# B&R Automation Studio project TD52 (part 65)

```c
  /* BusCreator: '<Root>/Bus Creator' incorporates:
   *  BusCreator: '<S1>/Bus Creator2'
   *  DataTypeConversion: '<S1>/Data Type Conversion19'
   *  DataTypeConversion: '<S1>/Data Type Conversion7'
   *  Outport: '<Root>/dbg'
   */
  Gen2_ref_Y->dbg.BDC.FF.wg_cd = (real32_T)r;
  Gen2_ref_Y->dbg.BDC.FF.u_tv_ff = (real32_T)rtb_Product4_d;

  /* MinMax: '<S490>/MinMax' incorporates:
   *  DataTypeConversion: '<S43>/Data Type Conversion25'
   */
  if ((Gen2_ref_B->BusInput3.bdcTv.rPos_min >= (real32_T)rtb_Switch_e) ||
      rtIsNaN((real32_T)rtb_Switch_e)) {
    rtb_Sum_mf = Gen2_ref_B->BusInput3.bdcTv.rPos_min;
  } else {
    rtb_Sum_mf = (real32_T)rtb_Switch_e;
  }

  /* End of MinMax: '<S490>/MinMax' */

  /* Logic: '<S426>/Logical Operator3' incorporates:
   *  Constant: '<S490>/Constant4'
   *  Logic: '<S426>/Logical Operator'
   *  Logic: '<S426>/Logical Operator2'
   *  Logic: '<S490>/Logical Operator1'
   *  Product: '<S490>/Divide'
   *  RelationalOperator: '<S490>/Relational Operator2'
   *  RelationalOperator: '<S490>/Relational Operator3'
   *  Sum: '<S490>/Sum'
   *  Sum: '<S490>/Sum2'
   *  UnitDelay: '<Root>/Unit Delay3'
   */
  rtb_LogicalOperator3_gq = (((Gen2_ref_DWork->UnitDelay3_DSTATE /
    rtb_deltafalllimit_ca >= 1.0 - rtb_PactOut) && (rtb_Divide3_ep <= rtb_Sum_mf
    + rtb_PactOut)) || (Gen2_ref_B->TP_ActSat_CBV.LogicalOperator1 &&
                        Gen2_ref_B->TP_ActSat_TV.LogicalOperator1) ||
    (!Gen2_ref_B->BusInput3.LR.bAct_CompActSatOnly));

  /* Switch: '<S491>/Switch3' incorporates:
   *  Constant: '<S426>/Constant'
   */
  if (rtb_bResetHlci) {
    rtb_LogicalOperator_aw = false;
  } else {
    /* Sum: '<S426>/Sum2' */
    rtb_Divide2_f = rtb_Switch_i5[0] - rtb_Switch_ks;

    /* Switch: '<S491>/Switch1' incorporates:
     *  Constant: '<S491>/FALSE'
     *  RelationalOperator: '<S491>/groesser '
     *  RelationalOperator: '<S491>/kleiner'
     *  UnitDelay: '<S491>/Unit Delay2'
     */
    if (rtb_Divide2_f < Gen2_ref_B->BusInput3.LR.rN_GasFlowSatComp_diffLo) {
      rtb_LogicalOperator_aw = false;
    } else {
      rtb_LogicalOperator_aw = ((rtb_Divide2_f >
        Gen2_ref_B->BusInput3.LR.rN_GasFlowSatComp_diffUp) ||
        Gen2_ref_DWork->UnitDelay2_DSTATE_j);
    }

    /* End of Switch: '<S491>/Switch1' */
  }

  /* End of Switch: '<S491>/Switch3' */

  /* Gain: '<S426>/Gain' */
  rtb_Sum_mf = 100000.0 * Gen2_ref_B->BusInput3.LR.rP2s_GasFlowSatComp_SettleLim;

  /* Outputs for Atomic SubSystem: '<S426>/TP' */
  /* RelationalOperator: '<S426>/Relational Operator' incorporates:
   *  SignalConversion generated from: '<S426>/Bus Selector3'
   */
  Gen2_ref_TP((rtb_Switch_i5[5] <= rtb_Sum_mf),
              Gen2_ref_B->BusInput3.LR.rTi_GasFlowSatComp_TP2psSettle,
              &Gen2_ref_B->TP, &Gen2_ref_DWork->TP, inst);

  /* End of Outputs for SubSystem: '<S426>/TP' */

  /* Outputs for Atomic SubSystem: '<S426>/TP1' */
  /* RelationalOperator: '<S426>/Relational Operator1' incorporates:
   *  SignalConversion generated from: '<S426>/Bus Selector5'
   */
  Gen2_ref_TP((rtb_Saturation >
               Gen2_ref_B->BusInput3.LR.rP_GasFlowSatComp_RotLim),
              Gen2_ref_B->BusInput3.LR.rTi_GasFlowSatComp_ProtTP,
              &Gen2_ref_B->TP1, &Gen2_ref_DWork->TP1, inst);

  /* End of Outputs for SubSystem: '<S426>/TP1' */

  /* Switch: '<S494>/etaVolConst' incorporates:
   *  Constant: '<S426>/Constant4'
   *  Logic: '<S426>/Logical Operator1'
   *  Logic: '<S426>/Logical Operator4'
   *  Switch: '<S426>/Switch'
   */
  if (rtb_bResetHlci) {
    rtb_Divide2_f = 1.0;
  } else if (Gen2_ref_B->BusInput3.LR.bActGasFlowSatComp &&
             rtb_LogicalOperator3_gq && rtb_LogicalOperator_aw &&
             (!Gen2_ref_B->TP.LogicalOperator1) &&
             Gen2_ref_B->TP1.LogicalOperator1) {
    /* Switch: '<S426>/Switch1' incorporates:
     *  Switch: '<S426>/Switch'
     */
    if (Gen2_ref_B->BusInput3.LR.bGS_GasFlowSatComp_active) {
      /* Switch: '<S426>/Switch2' */
      if (Gen2_ref_B->BusInput3.LR.bGS_GasFlowSatComp_UseProt) {
        rtb_Divide2_f = rtb_Saturation;
      } else {
        rtb_Divide2_f = rtb_kW2W1_h;
      }

      /* S-Function (sfix_look1_dyn): '<S426>/Lookup Table Dynamic' */
      /* Dynamic Look-Up Table Block: '<S426>/Lookup Table Dynamic'
       * Input0  Data Type:  Floating Point real_T
       * Input1  Data Type:  Floating Point real_T
       * Input2  Data Type:  Floating Point real_T
       * Output0 Data Type:  Floating Point real_T
       * Lookup Method: Linear_Endpoint
       *
       */
      LookUp_real_T_real_T( &(rtb_LookupTableDynamic_h),
                           &Gen2_ref_B->BusInput3.LR.rGainGasFlowSatComp_GS_y[0],
                           rtb_Divide2_f,
                           &Gen2_ref_B->BusInput3.LR.rGainGasFlowSatComp_GS_x[0],
                           7U, inst);
      rtb_Divide2_f = rtb_LookupTableDynamic_h;
    } else {
      rtb_Divide2_f = Gen2_ref_B->BusInput3.LR.rGainGasFlowSatComp;
    }
  } else {
    /* Switch: '<S426>/Switch' incorporates:
     *  Constant: '<S426>/Constant4'
     */
    rtb_Divide2_f = 1.0;
  }

  /* Delay: '<S494>/Delay' incorporates:
   *  Constant: '<S426>/Constant4'
   *  Delay: '<S425>/Delay'
   */
  Gen2_ref_DWork->icLoad_ir = ((((Gen2_ref_PrevZCSigState->Delay_Reset_ZCE_bc ==
    1) != (int32_T)rtb_bResetHlci) &&
    (Gen2_ref_PrevZCSigState->Delay_Reset_ZCE_bc != 3)) || rtb_bResetHlci ||
    Gen2_ref_DWork->icLoad_ir);
  Gen2_ref_PrevZCSigState->Delay_Reset_ZCE_bc = rtb_bResetHlci;
  if (Gen2_ref_DWork->icLoad_ir) {
    Gen2_ref_DWork->Delay_DSTATE_f = 1.0;
  }

  /* Sum: '<S494>/Difference Inputs1' incorporates:
   *  Delay: '<S494>/Delay'
   */
  rtb_Divide2_f -= Gen2_ref_DWork->Delay_DSTATE_f;

  /* Switch: '<S505>/Switch2' incorporates:
   *  RelationalOperator: '<S505>/LowerRelop1'
   */
  if (!(rtb_Divide2_f > rtb_Switch2_l)) {
    /* Switch: '<S505>/Switch' incorporates:
     *  RelationalOperator: '<S505>/UpperRelop'
     */
    if (rtb_Divide2_f < -10.0) {
      rtb_Switch2_l = -10.0;
    } else {
      rtb_Switch2_l = rtb_Divide2_f;
    }

    /* End of Switch: '<S505>/Switch' */
  }

  /* End of Switch: '<S505>/Switch2' */

  /* Sum: '<S494>/Difference Inputs2' incorporates:
   *  Delay: '<S494>/Delay'
   */
  rtb_Switch2_l += Gen2_ref_DWork->Delay_DSTATE_f;

  /* Switch: '<Root>/GasStop' incorporates:
   *  Constant: '<Root>/Constant3'
   *  Product: '<S5>/Product'
   */
  if (rtb_dbg_HLCi) {
    rtb_Sum_c = 0.0;
  } else {
    rtb_Sum_c = Gen2_ref_B->sf_IntegerZOH_f.y * rtb_Switch2_l;
  }

  /* End of Switch: '<Root>/GasStop' */

  /* Outputs for Atomic SubSystem: '<S268>/Mg' */
  Gen2_ref_Mg(Gen2_ref_B->BusInput3.eng.rRho_gas_M, &Gen2_ref_B->Mg_l, inst);

  /* End of Outputs for SubSystem: '<S268>/Mg' */

  /* Outputs for Atomic SubSystem: '<S268>/lam2cg' */
  Gen2_ref_lam2cg1(rtb_Product1_fu,
                   Gen2_ref_B->BusInput3.eng.rMin_Air_Ratio_M_kg,
                   &Gen2_ref_B->lam2cg_i, inst);

  /* End of Outputs for SubSystem: '<S268>/lam2cg' */

  /* Product: '<S268>/Divide3' incorporates:
   *  Bias: '<S268>/Bias'
   *  Constant: '<S268>/R_air'
   *  Product: '<S268>/Divide2'
   */
  rtb_Switch_ks = (Gen2_ref_B->Mg_l.Bias * Gen2_ref_B->lam2cg_i.Divide + 1.0) *
    287.15;

  /* Product: '<S268>/Divide' incorporates:
   *  Product: '<S268>/Divide3'
   */
  rtb_Divide_ab[0] = rtb_SumofElements_l / rtb_Switch_ks *
    Gen2_ref_B->BusInput3.fdc.rCF[0];
  rtb_Divide_ab[1] = rtb_RoundingFunction / rtb_Switch_ks *
    Gen2_ref_B->BusInput3.fdc.rCF[1];
  rtb_Divide_ab[2] = rtb_Switch2_d1 / rtb_Switch_ks *
    Gen2_ref_B->BusInput3.fdc.rCF[2];
  rtb_Divide_ab[3] = rtb_Product1_mqz / rtb_Switch_ks *
    Gen2_ref_B->BusInput3.fdc.rCF[3];

  /* Product: '<S268>/Divide1' incorporates:
   *  Sum: '<S268>/Sum of Elements'
   */
  rtb_Sum_mf = (((rtb_Divide_ab[0] + rtb_Divide_ab[1]) + rtb_Divide_ab[2]) +
                rtb_Divide_ab[3]) * Gen2_ref_B->lam2cg_i.Divide;

  /* Switch: '<S268>/Switch' incorporates:
   *  Constant: '<S268>/Constant5'
   */
  if (Gen2_ref_B->BusInput3.fdc.bActive_dyn) {
    rtb_Divide2_f = rtb_Sum_mf;
  } else {
    rtb_Divide2_f = 0.0;
  }

  /* End of Switch: '<S268>/Switch' */

  /* Abs: '<S289>/Abs' incorporates:
   *  Abs: '<S817>/Abs'
   */
  delta_y = rtb_bResetHlci_0;
  rtb_Sum2_a1 = delta_y;

  /* Switch: '<S289>/Switch' incorporates:
   *  Constant: '<S289>/Constant2'
   *  RelationalOperator: '<S289>/Relational Operator'
   */
  if (1.0 >= rtb_Sum2_a1) {
    rtb_SumofElements_l = 1.0;
  } else {
    rtb_SumofElements_l = Gen2_ref_B->T2s_filt.Switch;
  }

  /* End of Switch: '<S289>/Switch' */

  /* Outputs for Atomic SubSystem: '<S268>/lam2cg1' */
  Gen2_ref_lam2cg1_a(rtb_Product1_fu, Gen2_ref_B->BusInput3.eng.rMin_Air_Ratio_M,
                     &Gen2_ref_B->lam2cg1_i, inst);

  /* End of Outputs for SubSystem: '<S268>/lam2cg1' */

  /* Gain: '<S268>/Gain2' */
  rtb_Sum2_a1 = rtb_Gain_kp;

  /* Product: '<S268>/Product3' incorporates:
   *  Gain: '<S268>/StandardCond'
   *  Product: '<S268>/Divide10'
   *  Product: '<S268>/Divide8'
   */
  rtb_Sum2_a1 = rtb_Switch4_p / rtb_SumofElements_l * 0.0026957809030347889 *
    rtb_Sum_e * Gen2_ref_B->lam2cg1_i.Divide * rtb_Sum2_a1 *
    Gen2_ref_B->BusInput3.eng.rRho_gas_M;

  /* Sum: '<S268>/Add1' */
  rtb_SumofElements_l = rtb_Divide2_f + rtb_Sum2_a1;

  /* MATLAB Function: '<S5>/IntegerZOH1' incorporates:
   *  Product: '<S5>/Divide1'
   */
  Gen2_ref_IntegerZOH(Gen2_ref_B->BusInput.IN_EC_rGT_RatioMix_TC2 *
                      rtb_SumofElements_l, Npred, &Gen2_ref_B->sf_IntegerZOH1_n,
                      &Gen2_ref_DWork->sf_IntegerZOH1_n, inst);

  /* Switch: '<Root>/GasStop2' incorporates:
   *  Constant: '<Root>/Constant3'
   *  Product: '<S5>/Product1'
   */
  if (rtb_dbg_HLCi) {
    rtb_Switch2_jq = 0.0;
  } else {
    rtb_Switch2_jq = rtb_Switch2_l * Gen2_ref_B->sf_IntegerZOH1_n.y;
  }

  /* End of Switch: '<Root>/GasStop2' */

  /* Switch: '<S1>/Switch1' incorporates:
   *  Constant: '<S1>/Constant3'
   *  Constant: '<S30>/Constant'
   *  RelationalOperator: '<S30>/Compare'
   */
  if (Gen2_ref_B->BusInput3.eng.rNum_TV > 0.5) {
    /* Outputs for Atomic SubSystem: '<S45>/Linearization' */
    /* S-Function (sfix_look1_dyn): '<S166>/LCRScal_Lam_EOT1' */
    /* Dynamic Look-Up Table Block: '<S166>/LCRScal_Lam_EOT1'
     * Input0  Data Type:  Floating Point real_T
     * Input1  Data Type:  Floating Point real_T
     * Input2  Data Type:  Floating Point real_T
     * Output0 Data Type:  Floating Point real_T
     * Lookup Method: Linear_Endpoint
     *
     */
    LookUp_real_T_real_T( &(rtb_LCRScal_Lam_EOT1),
                         &Gen2_ref_B->BusInput3.bdcTv.rPosTv_Lin_y[0],
                         rtb_Switch2_by,
                         &Gen2_ref_B->BusInput3.bdcTv.rPosTv_Lin_x[0], 9U, inst);

    /* End of Outputs for SubSystem: '<S45>/Linearization' */
    rtb_Switch13 = rtb_LCRScal_Lam_EOT1;
  } else {
    rtb_Switch13 = 1.0;
  }

  /* End of Switch: '<S1>/Switch1' */

  /* Switch: '<S1>/Switch12' incorporates:
   *  Constant: '<S1>/Constant1'
   *  Logic: '<S1>/Logical Operator6'
   *  Logic: '<S1>/Logical Operator8'
   */
  if ((!Gen2_ref_B->BusInput3.bdcMisc.bSwitchOutputSampleSS) ||
      Gen2_ref_B->TON2.LogicalOperator3) {
    Npred = Gen2_ref_B->BusInput3.bdcMisc.iOutputSample;
  } else {
    Npred = 1;
  }

  /* End of Switch: '<S1>/Switch12' */

  /* MATLAB Function: '<S1>/IntegerZOH' */
  Gen2_ref_IntegerZOH(rtb_Switch13, Npred, &Gen2_ref_B->sf_IntegerZOH,
                      &Gen2_ref_DWork->sf_IntegerZOH, inst);

  /* Switch: '<S1>/Switch3' incorporates:
   *  Constant: '<S1>/Constant'
   *  Constant: '<S29>/Constant'
   *  RelationalOperator: '<S29>/Compare'
   */
  if (Gen2_ref_B->BusInput3.eng.rNum_CBV > 1.5) {
    /* Switch: '<S1>/Switch5' */
    if (Gen2_ref_B->BusInput3.bdcCbv.bFFonly_2nd_CBV) {
      rtb_Product4_d = rtb_Sum1_lo;
    } else {
      rtb_Product4_d = rtb_Switch1_kk;
    }

    /* End of Switch: '<S1>/Switch5' */
  } else {
    rtb_Product4_d = 0.0;
  }

  /* End of Switch: '<S1>/Switch3' */

  /* Switch: '<S1>/Switch4' incorporates:
   *  Constant: '<S1>/Constant'
   *  Constant: '<S28>/Constant'
   *  RelationalOperator: '<S28>/Compare'
   */
  if (Gen2_ref_B->BusInput3.eng.rNum_CBV > 2.5) {
    /* Switch: '<S1>/Switch6' */
    if (Gen2_ref_B->BusInput3.bdcCbv.bFFonly_3rd_CBV) {
      rtb_MinMax_a = rtb_Sum1_lo;
    } else {
      rtb_MinMax_a = rtb_Switch1_kk;
    }

    /* End of Switch: '<S1>/Switch6' */
  } else {
    rtb_MinMax_a = 0.0;
  }

  /* End of Switch: '<S1>/Switch4' */

  /* SignalConversion generated from: '<S38>/ SFunction ' incorporates:
   *  MATLAB Function: '<S1>/IntegerZOH1'
   */
  rtb_TmpSignalConversionAtSFun_p[0] = rtb_Switch1_kk;
  rtb_TmpSignalConversionAtSFun_p[1] = rtb_Product4_d;
  rtb_TmpSignalConversionAtSFun_p[2] = rtb_MinMax_a;

  /* MATLAB Function: '<S1>/IntegerZOH1' incorporates:
   *  SignalConversion generated from: '<S38>/ SFunction '
   */
  if (!Gen2_ref_DWork->count_not_empty) {
    Gen2_ref_DWork->count_not_empty = true;
    Gen2_ref_DWork->u_z[0] = rtb_Switch1_kk;
    Gen2_ref_DWork->u_z[1] = rtb_Product4_d;
    Gen2_ref_DWork->u_z[2] = rtb_MinMax_a;
  }

  if (Gen2_ref_DWork->count_p < Npred) {
    rtb_TmpSignalConversionAtSFun_p[0] = Gen2_ref_DWork->u_z[0];
    rtb_TmpSignalConversionAtSFun_p[1] = Gen2_ref_DWork->u_z[1];
    rtb_TmpSignalConversionAtSFun_p[2] = Gen2_ref_DWork->u_z[2];
    Gen2_ref_DWork->count_p++;
  } else {
    Gen2_ref_DWork->u_z[0] = rtb_Switch1_kk;
    Gen2_ref_DWork->u_z[1] = rtb_Product4_d;
    Gen2_ref_DWork->u_z[2] = rtb_MinMax_a;
    Gen2_ref_DWork->count_p = 1.0;
  }

  /* S-Function (sfix_look1_dyn): '<S46>/Lookup Table Dynamic' */
  /* Dynamic Look-Up Table Block: '<S46>/Lookup Table Dynamic'
   * Input0  Data Type:  Floating Point real_T
   * Input1  Data Type:  Floating Point real_T
   * Input2  Data Type:  Floating Point real_T
   * Output0 Data Type:  Floating Point real_T
   * Lookup Method: Linear_Endpoint
   *
   */
  LookUp_real_T_real_T( &(rtb_Divide2_f),
                       &Gen2_ref_B->BusInput3.bdcWgv.rCd_vect_x[0], r,
                       &Gen2_ref_B->BusInput3.bdcWgv.rCd_vect_y[0], 10U, inst);

  /* MinMax: '<S46>/MinMax' */
  r = Gen2_ref_B->BusInput3.bdcWgv.rCd_vect_x[0];
  for (k = 0; k < 10; k++) {
    u1 = Gen2_ref_B->BusInput3.bdcWgv.rCd_vect_x[k + 1];
    if ((!(r >= u1)) && (!rtIsNaN(u1))) {
      r = u1;
    }
  }

  /* End of MinMax: '<S46>/MinMax' */

  /* Abs: '<S170>/Abs' */
  rtb_Product4_d = fabs(r);

  /* Switch: '<S170>/Switch' incorporates:
   *  Constant: '<S170>/Constant2'
   *  RelationalOperator: '<S170>/Relational Operator'
   */
  if (2.2204460492503131E-16 >= rtb_Product4_d) {
    rtb_Sum_e = 2.2204460492503131E-16;
  } else {
    rtb_Sum_e = r;
  }

  /* End of Switch: '<S170>/Switch' */

  /* Saturate: '<S46>/Saturation3' */
  if (Gen2_ref_B->BusInput3.eng.rNum_WGV > 1.0) {
    r = 1.0;
  } else if (Gen2_ref_B->BusInput3.eng.rNum_WGV < 0.0) {
    r = 0.0;
  } else {
    r = Gen2_ref_B->BusInput3.eng.rNum_WGV;
  }

  /* End of Saturate: '<S46>/Saturation3' */

  /* Product: '<S46>/Divide2' incorporates:
   *  Product: '<S46>/Divide'
   */
  rtb_Switch2_by = rtb_Divide2_f / rtb_Sum_e * r;

  /* Switch: '<S1>/Switch2' incorporates:
   *  Constant: '<S1>/max_PR2'
   */
  if (Gen2_ref_B->BusInput3.bdcWgv.bTransWGctrl_FF) {
    r = rtb_Switch2_by;
  } else {
    r = 0.0;
  }

  /* End of Switch: '<S1>/Switch2' */

  /* Outputs for Atomic SubSystem: '<S192>/N_TC_LP_filt' */
  /* DataTypeConversion: '<S4>/Data Type Conversion20' */
  Gen2_ref_N_TC_HP_filt((real_T)Gen2_ref_B->BusInput.rN_TC_LP,
                        Gen2_ref_B->BusInput3.inFilt.rTiF_N, rtb_bResetBdc,
                        &Gen2_ref_B->N_TC_LP_filt, &Gen2_ref_DWork->N_TC_LP_filt, inst);

  /* End of Outputs for SubSystem: '<S192>/N_TC_LP_filt' */

  /* Sum: '<S22>/Sum1' */
  rtb_Divide2_f = Gen2_ref_B->N_TC_LP_filt.Switch -
    Gen2_ref_B->BusInput3.bdcWgv.rTcMaxSpeed;

  /* Gain: '<S22>/Gain' */
  rtb_Gain_kp = 0.001 * rtb_Divide2_f;

  /* DiscreteIntegrator: '<S22>/Discrete-Time Integrator' */
  if (rtb_LogicalOperator2_dc ||
      (Gen2_ref_DWork->DiscreteTimeIntegrator_PrevR_jc != 0)) {
    Gen2_ref_DWork->DiscreteTimeIntegrator_DSTATE_i = 0.0;
  }

  if (Gen2_ref_DWork->DiscreteTimeIntegrator_DSTATE_i >= 1.0) {
    Gen2_ref_DWork->DiscreteTimeIntegrator_DSTATE_i = 1.0;
  } else if (Gen2_ref_DWork->DiscreteTimeIntegrator_DSTATE_i <= 0.0) {
    Gen2_ref_DWork->DiscreteTimeIntegrator_DSTATE_i = 0.0;
  }

  /* Switch: '<S22>/Switch' incorporates:
   *  Constant: '<S22>/ON1'
   */
  if (Gen2_ref_B->BusInput3.bdcWgv.bWgvTcOvrspdCtrl) {
    /* Sum: '<S22>/Sum3' incorporates:
     *  DiscreteIntegrator: '<S22>/Discrete-Time Integrator'
     *  Product: '<S22>/Product'
     */
    rtb_Divide2_f = rtb_Gain_kp *
      Gen2_ref_B->BusInput3.bdcWgv.rKpWgvTcOvrspdCtrl +
      Gen2_ref_DWork->DiscreteTimeIntegrator_DSTATE_i;

    /* Saturate: '<S22>/Saturation' */
    if (rtb_Divide2_f > 1.0) {
      rtb_Divide2_f = 1.0;
    } else if (rtb_Divide2_f < 0.0) {
      rtb_Divide2_f = 0.0;
    }

    /* End of Saturate: '<S22>/Saturation' */
  } else {
    rtb_Divide2_f = 0.0;
  }

  /* End of Switch: '<S22>/Switch' */

  /* Sum: '<S22>/Sum' */
  rtb_Divide2_f += r;

  /* Switch: '<S42>/Switch2' incorporates:
   *  RelationalOperator: '<S42>/LowerRelop1'
   *  RelationalOperator: '<S42>/UpperRelop'
   *  Switch: '<S42>/Switch'
   */
  if (rtb_Divide2_f > Gen2_ref_B->BusInput3.bdcWgv.rPos_max) {
    rtb_Divide2_f = Gen2_ref_B->BusInput3.bdcWgv.rPos_max;
  } else if (rtb_Divide2_f < Gen2_ref_B->BusInput3.bdcWgv.rPos_min) {
    /* Switch: '<S42>/Switch' */
    rtb_Divide2_f = Gen2_ref_B->BusInput3.bdcWgv.rPos_min;
  }

  /* End of Switch: '<S42>/Switch2' */

  /* MATLAB Function: '<S1>/IntegerZOH2' */
  Gen2_ref_IntegerZOH(rtb_Divide2_f, Npred, &Gen2_ref_B->sf_IntegerZOH2,
                      &Gen2_ref_DWork->sf_IntegerZOH2, inst);

  /* Switch: '<Root>/BDC_traj1' incorporates:
   *  Switch: '<Root>/BDC_traj2'
   */
  if (rtb_LogicalOperator) {
    rtb_Divide2_f = rtb_TmpSignalConversionAtSFun_p[0];
    r = rtb_TmpSignalConversionAtSFun_p[0];
  } else {
    rtb_Divide2_f = rtb_TmpSignalConversionAtSFun_p[1];
    r = rtb_TmpSignalConversionAtSFun_p[2];
  }

  /* End of Switch: '<Root>/BDC_traj1' */

  /* Logic: '<S16>/Logical Operator6' */
  rtb_bCBV_min = !Gen2_ref_B->BusInput3.inFilt.bFiltOutput;

  /* SignalConversion generated from: '<S873>/ SFunction ' incorporates:
   *  MATLAB Function: '<S16>/FILTER no delay'
   */
  rtb_Switch_g[0] = rtb_Sum_c;
  rtb_Switch_g[1] = rtb_Switch2_jq;
  rtb_Switch_g[2] = rtb_Product1_fu;
  rtb_Switch_g[3] = Gen2_ref_B->sf_IntegerZOH.y;
  rtb_Switch_g[4] = rtb_TmpSignalConversionAtSFun_p[0];
  rtb_Switch_g[5] = Gen2_ref_B->sf_IntegerZOH2.y;
  rtb_Switch_g[6] = rtb_Divide2_f;
  rtb_Switch_g[7] = r;

  /* MATLAB Function: '<S16>/FILTER no delay' incorporates:
   *  Logic: '<S16>/Logical Operator1'
   */
  if ((!Gen2_ref_DWork->x_not_empty) || (rtb_bCBV_min || rtb_bResetBdc)) {
    for (i = 0; i < 8; i++) {
      Gen2_ref_DWork->x[i] = rtb_Switch_g[i];
    }

    Gen2_ref_DWork->x_not_empty = true;
  }

  if (Gen2_ref_B->BusInput3.eng.Ts > 0.0) {
    if ((Gen2_ref_B->BusInput3.inFilt.rTiF_OUT >= Gen2_ref_B->BusInput3.eng.Ts) ||
        rtIsNaN(Gen2_ref_B->BusInput3.eng.Ts)) {
      rtb_Product4_d = Gen2_ref_B->BusInput3.inFilt.rTiF_OUT;
    } else {
      rtb_Product4_d = Gen2_ref_B->BusInput3.eng.Ts;
    }

    for (i = 0; i < 8; i++) {
      Gen2_ref_DWork->x[i] += (rtb_Switch_g[i] - Gen2_ref_DWork->x[i]) /
        rtb_Product4_d * Gen2_ref_B->BusInput3.eng.Ts;
      rtb_Switch_g[i] = Gen2_ref_DWork->x[i];
    }
  } else {
    for (i = 0; i < 8; i++) {
      Gen2_ref_DWork->x[i] = rtb_Switch_g[i];
    }
  }

  /* Switch: '<S16>/Switch' */
  rtb_Sum_og[0] = rtb_Sum_c;
  rtb_Sum_og[1] = rtb_Switch2_jq;
  rtb_Sum_og[2] = rtb_Product1_fu;
  rtb_Sum_og[3] = Gen2_ref_B->sf_IntegerZOH.y;
  rtb_Sum_og[4] = rtb_TmpSignalConversionAtSFun_p[0];
  rtb_Sum_og[5] = Gen2_ref_B->sf_IntegerZOH2.y;
  rtb_Sum_og[6] = rtb_Divide2_f;
  rtb_Sum_og[7] = r;
  for (i = 0; i < 8; i++) {
    rtb_Divide2_f = rtb_Switch_g[i];
    if (rtb_bCBV_min) {
      rtb_Divide2_f = rtb_Sum_og[i];
    }

    rtb_Switch_g[i] = rtb_Divide2_f;
  }

  /* End of Switch: '<S16>/Switch' */

  /* Gain: '<S430>/bar2mbar1' */
  r = rtb_mbar2pa_i;

  /* Sum: '<S8>/Sum' */
  rtb_Divide2_f = rtb_Product1_c1_tmp;

  /* Switch: '<S422>/Switch' incorporates:
   *  Constant: '<S422>/Constant4'
   *  Logic: '<S422>/Logical Operator2'
   *  RelationalOperator: '<S422>/Relational Operator'
   */
  if ((rtb_Divide2_f > Gen2_ref_B->BusInput3.SpeedCtrl.rOutOfNWindow) &&
      Gen2_ref_B->BusInput3.SpeedCtrl.bScaleLeanoxErrorEnrichment) {
    /* Product: '<S422>/Product8' incorporates:
     *  Constant: '<S422>/Constant'
     *  DataTypeConversion: '<S4>/Data Type Conversion28'
     *  Product: '<S422>/Product5'
     *  Sum: '<S14>/Sum10'
     *  Sum: '<S422>/Sum3'
     *  Sum: '<S8>/Sum2'
     */
    rtb_Divide2_f = (((Gen2_ref_B->BusInput.rOffsetLamLimit + rtb_PactOut_o) +
                      rtb_Sum4_ny) * rtb_Sum1_idx_2 + 1.0) * rtb_Switch_i5[0];

    /* Saturate: '<S422>/Saturation1' */
    if (rtb_Divide2_f <= 1.0) {
      rtb_Divide2_f = 1.0;
    }

    /* End of Saturate: '<S422>/Saturation1' */

    /* Product: '<S422>/Divide' incorporates:
     *  Constant: '<S422>/Constant'
     *  Product: '<S422>/Product3'
     *  Product: '<S422>/Product7'
     *  Sum: '<S422>/Sum2'
     */
    rtb_Divide2_f = (rtb_Sum2_kg * rtb_Sum1_idx_2 + 1.0) *
      Gen2_ref_B->BusInput3.eng.rN_Nom / rtb_Divide2_f;

    /* Saturate: '<S422>/Saturation' */
    if (rtb_Divide2_f > 1.0) {
      rtb_Divide2_f = 1.0;
    } else if (rtb_Divide2_f < 0.1) {
      rtb_Divide2_f = 0.1;
    }

    /* End of Saturate: '<S422>/Saturation' */
  } else {
    rtb_Divide2_f = 1.0;
  }

  /* End of Switch: '<S422>/Switch' */

  /* Product: '<S8>/Product' */
  rtb_Product4_d = rtb_Gain1_fr * Gen2_ref_B->BusInput3.SpeedCtrl.rFactProt;

  /* Gain: '<S423>/W2kW' incorporates:
   *  Sum: '<S8>/Sum1'
   */
  rtb_Sum4_ny = (rtb_Switch_i5[3] - rtb_Product4_d) * 0.001;

  /* Switch: '<S476>/Switch2' incorporates:
   *  RelationalOperator: '<S476>/LowerRelop1'
   */
  if (rtb_Sum4_ny > Gen2_ref_B->BusInput3.eng.rP_Nom) {
    rtb_Sum_c = Gen2_ref_B->BusInput3.eng.rP_Nom;
  } else {
    /* Product: '<S473>/Divide6' */
    rtb_Sum_c = Gen2_ref_B->BusInput3.eng.rP_Nom *
      Gen2_ref_B->BusInput3.leanox.rP_P2sRedIP_SP_Norm;

    /* Switch: '<S476>/Switch' incorporates:
     *  RelationalOperator: '<S476>/UpperRelop'
     */
    if (!(rtb_Sum4_ny < rtb_Sum_c)) {
      rtb_Sum_c = rtb_Sum4_ny;
    }

    /* End of Switch: '<S476>/Switch' */
  }

  /* End of Switch: '<S476>/Switch2' */

  /* MATLAB Function: '<S473>/2-point interpolation, with extrapolation' */
  upointinterpolationwithextrapol(rtb_Sum_c,
    Gen2_ref_B->BusInput3.leanox.Comp_IgnP_x,
    Gen2_ref_B->BusInput3.leanox.Comp_IgnP_y,
    &Gen2_ref_B->sf_2pointinterpolationwithext_j, inst);

  /* Switch: '<S473>/Switch1' incorporates:
   *  Constant: '<S473>/Pel_a (kW)1'
   *  DataTypeConversion: '<S4>/Data Type Conversion22'
   *  Product: '<S473>/Divide5'
   *  Sum: '<S473>/Add12'
   */
  if (Gen2_ref_B->BusInput3.leanox.bZZPKorr) {
    rtb_Product4_d = (Gen2_ref_B->BusInput.rCA_Ign_OP_Power -
                      Gen2_ref_B->N_TC_HP_filt.Switch) *
      Gen2_ref_B->sf_2pointinterpolationwithext_j.y;
  } else {
    rtb_Product4_d = 0.0;
  }

  /* End of Switch: '<S473>/Switch1' */

  /* Switch: '<S477>/Switch2' incorporates:
   *  RelationalOperator: '<S477>/LowerRelop1'
   */
  if (rtb_Sum4_ny > Gen2_ref_B->BusInput3.eng.rP_Nom) {
    rtb_Sum_c = Gen2_ref_B->BusInput3.eng.rP_Nom;
  } else {
    /* Product: '<S473>/Divide1' */
    rtb_Sum_c = Gen2_ref_B->BusInput3.eng.rP_Nom *
      Gen2_ref_B->BusInput3.leanox.rP2s_Comp_Act_SP;

    /* Switch: '<S477>/Switch' incorporates:
     *  RelationalOperator: '<S477>/UpperRelop'
     */
    if (!(rtb_Sum4_ny < rtb_Sum_c)) {
      rtb_Sum_c = rtb_Sum4_ny;
    }

    /* End of Switch: '<S477>/Switch' */
  }

  /* End of Switch: '<S477>/Switch2' */

  /* MATLAB Function: '<S473>/2-point interpolation, with extrapolation1' */
  upointinterpolationwithextrapol(rtb_Sum_c,
    Gen2_ref_B->BusInput3.leanox.Comp_ChTmp_x,
    Gen2_ref_B->BusInput3.leanox.Comp_ChTmp_y,
    &Gen2_ref_B->sf_2pointinterpolationwithext_o, inst);

  /* Switch: '<S473>/Switch3' incorporates:
   *  Constant: '<S473>/Pel_a (kW)3'
   */
  if (Gen2_ref_B->BusInput3.leanox.bHum_Act) {
    rtb_Sum1_dh = Gen2_ref_B->BusInput3.leanox.rP2s_Comp_HumOffset;
  } else {
    rtb_Sum1_dh = 0.0;
  }

  /* End of Switch: '<S473>/Switch3' */

  /* Switch: '<S473>/Switch2' incorporates:
   *  Constant: '<S473>/Pel_a (kW)2'
   *  Product: '<S473>/Divide9'
   *  Sum: '<S473>/Add13'
   */
  if (Gen2_ref_B->BusInput3.leanox.bt2Korr) {
    rtb_bResetHlci_0 = (Gen2_ref_B->T2s_filt.Switch -
                        Gen2_ref_B->BusInput3.leanox.rT_2) *
      Gen2_ref_B->sf_2pointinterpolationwithext_o.y;
  } else {
    rtb_bResetHlci_0 = 0.0;
  }

  /* End of Switch: '<S473>/Switch2' */

  /* Sum: '<S459>/Add11' */
  rtb_Sum_c = (rtb_Product4_d + rtb_bResetHlci_0) + rtb_Sum1_dh;

  /* Switch: '<S423>/Switch1' incorporates:
   *  Product: '<S423>/Divide6'
   *  Sum: '<S423>/Add4'
   */
  if (Gen2_ref_B->BusInput.tLEANOXin.bZylAusfall) {
    /* Switch: '<S455>/Switch' incorporates:
     *  Abs: '<S455>/Abs'
     *  Constant: '<S455>/Constant2'
     *  RelationalOperator: '<S455>/Relational Operator'
     */
    if (1.0 >= fabs(Gen2_ref_B->BusInput3.eng.rNum_Cyl_Eng)) {
      rtb_bResetHlci_0 = 1.0;
    } else {
      rtb_bResetHlci_0 = Gen2_ref_B->BusInput3.eng.rNum_Cyl_Eng;
    }

    /* End of Switch: '<S455>/Switch' */
    rtb_Switch2_jq = rtb_Sum4_ny / rtb_bResetHlci_0 + rtb_Sum4_ny;
  } else {
    rtb_Switch2_jq = rtb_Sum4_ny;
  }

  /* End of Switch: '<S423>/Switch1' */

  /* Abs: '<S446>/Abs' */
  rtb_Product4_d = fabs(rtb_Switch_i5[0]);

  /* Switch: '<S446>/Switch' incorporates:
   *  Constant: '<S446>/Constant2'
   *  RelationalOperator: '<S446>/Relational Operator'
   */
  if (1.0 >= rtb_Product4_d) {
    rtb_MinMax_a = 1.0;
  } else {
    rtb_MinMax_a = rtb_Switch_i5[0];
  }

  /* End of Switch: '<S446>/Switch' */

  /* Switch: '<S423>/Switch4' */
  if (Gen2_ref_B->BusInput3.leanox.bLp_c_Ena) {
    rtb_Product4_d = Gen2_ref_B->BusInput3.leanox.rP_c;
  } else {
    rtb_Product4_d = Gen2_ref_B->BusInput3.leanox.rP_1;
  }

  /* End of Switch: '<S423>/Switch4' */

  /* Switch: '<S423>/Switch2' incorporates:
   *  Logic: '<S423>/Logical Operator1'
   *  Product: '<S423>/Divide4'
   *  RelationalOperator: '<S423>/Relational Operator1'
   *  RelationalOperator: '<S423>/Relational Operator3'
   *  Sum: '<S423>/Add5'
   *  Switch: '<S423>/Switch5'
   */
  if (rtb_Switch2_jq < rtb_Product4_d) {
    /* Switch: '<S423>/Switch_b_c' incorporates:
     *  Logic: '<S423>/Logical Operator'
     *  RelationalOperator: '<S423>/Relational Operator2'
     */
    if (Gen2_ref_B->BusInput3.leanox.bLp_c_Ena && (rtb_Switch2_jq <
         Gen2_ref_B->BusInput3.leanox.rP_c)) {
      /* SignalConversion generated from: '<S423>/Lookup Table Dynamic1' */
      rtb_TmpSignalConversionAtLoo_ht[0] =
        Gen2_ref_B->BusInput3.leanox.rPr_mbar_0;

      /* Switch: '<S456>/Switch' incorporates:
       *  Abs: '<S456>/Abs'
       *  Constant: '<S456>/Constant2'
       *  RelationalOperator: '<S456>/Relational Operator'
       */
      if (1.0 >= fabs(Gen2_ref_B->BusInput3.leanox.rT_c)) {
        rtb_bResetHlci_0 = 1.0;
      } else {
        rtb_bResetHlci_0 = Gen2_ref_B->BusInput3.leanox.rT_c;
      }

      /* End of Switch: '<S456>/Switch' */

      /* SignalConversion generated from: '<S423>/Lookup Table Dynamic1' incorporates:
       *  Product: '<S423>/Divide5'
       */
      rtb_TmpSignalConversionAtLoo_ht[1] =
        Gen2_ref_B->BusInput3.leanox.rPr_mbar_c *
        Gen2_ref_B->BusInput3.leanox.rN_c / rtb_bResetHlci_0 *
        Gen2_ref_B->T2s_filt.Switch / rtb_MinMax_a;

      /* SignalConversion generated from: '<S423>/Lookup Table Dynamic1' incorporates:
       *  Constant: '<S423>/Pel_a (kW)1'
       */
      rtb_TmpSignalConversionAtLook_d[0] = 0.0;
      rtb_TmpSignalConversionAtLook_d[1] = Gen2_ref_B->BusInput3.leanox.rP_c;

      /* S-Function (sfix_look1_dyn): '<S423>/Lookup Table Dynamic1' */
      /* Dynamic Look-Up Table Block: '<S423>/Lookup Table Dynamic1'
       * Input0  Data Type:  Floating Point real_T
       * Input1  Data Type:  Floating Point real_T
       * Input2  Data Type:  Floating Point real_T
       * Output0 Data Type:  Floating Point real_T
       * Lookup Method: Linear_Endpoint
       *
       */
      LookUp_real_T_real_T( &(rtb_LookupTableDynamic1_o),
                           &rtb_TmpSignalConversionAtLoo_ht[0], rtb_Switch2_jq,
                           &rtb_TmpSignalConversionAtLook_d[0], 1U, inst);
      rtb_Product4_d = rtb_LookupTableDynamic1_o;
    } else {
      /* SignalConversion generated from: '<S423>/Lookup Table Dynamic' */
      rtb_TmpSignalConversionAtLoo_ht[0] =
        Gen2_ref_B->BusInput3.leanox.rPr_mbar_0;

      /* Switch: '<S454>/Switch' incorporates:
       *  Abs: '<S454>/Abs'
       *  Constant: '<S454>/Constant2'
       *  RelationalOperator: '<S454>/Relational Operator'
       */
      if (1.0 >= fabs(Gen2_ref_B->BusInput3.leanox.rT_1)) {
        rtb_bResetHlci_0 = 1.0;
      } else {
        rtb_bResetHlci_0 = Gen2_ref_B->BusInput3.leanox.rT_1;
      }

      /* End of Switch: '<S454>/Switch' */

      /* SignalConversion generated from: '<S423>/Lookup Table Dynamic' incorporates:
       *  Product: '<S423>/Divide1'
       */
      rtb_TmpSignalConversionAtLoo_ht[1] =
        Gen2_ref_B->BusInput3.leanox.rPr_mbar_1 *
        Gen2_ref_B->BusInput3.leanox.rN_1 / rtb_bResetHlci_0 *
        Gen2_ref_B->T2s_filt.Switch / rtb_MinMax_a;

      /* SignalConversion generated from: '<S423>/Lookup Table Dynamic' incorporates:
       *  Constant: '<S423>/Pel_a (kW)3'
       */
      rtb_TmpSignalConversionAtLook_d[0] = 0.0;
      rtb_TmpSignalConversionAtLook_d[1] = Gen2_ref_B->BusInput3.leanox.rP_1;

      /* S-Function (sfix_look1_dyn): '<S423>/Lookup Table Dynamic' */
      /* Dynamic Look-Up Table Block: '<S423>/Lookup Table Dynamic'
       * Input0  Data Type:  Floating Point real_T
       * Input1  Data Type:  Floating Point real_T
       * Input2  Data Type:  Floating Point real_T
       * Output0 Data Type:  Floating Point real_T
       * Lookup Method: Linear_Endpoint
       *
       */
      LookUp_real_T_real_T( &(rtb_LookupTableDynamic_nk),
                           &rtb_TmpSignalConversionAtLoo_ht[0], rtb_Switch2_jq,
                           &rtb_TmpSignalConversionAtLook_d[0], 1U, inst);
      rtb_Product4_d = rtb_LookupTableDynamic_nk;
    }

    /* End of Switch: '<S423>/Switch_b_c' */
  } else {
    if (Gen2_ref_B->BusInput3.leanox.bLp_c_Ena && (rtb_Switch2_jq <
         Gen2_ref_B->BusInput3.leanox.rP_1)) {
      /* Sum: '<S423>/Add1' incorporates:
       *  Switch: '<S423>/Switch5'
       */
      rtb_Product4_d = Gen2_ref_B->BusInput3.leanox.rP_1 -
        Gen2_ref_B->BusInput3.leanox.rP_c;

      /* Sum: '<S423>/Sum4' incorporates:
       *  Switch: '<S423>/Switch5'
       */
      rtb_Sum1_dh = Gen2_ref_B->BusInput3.leanox.rP_c +
        Gen2_ref_B->BusInput3.leanox.rP_Eng_Frict;

      /* Switch: '<S449>/Switch' incorporates:
       *  Abs: '<S449>/Abs'
       *  Constant: '<S449>/Constant2'
       *  RelationalOperator: '<S449>/Relational Operator'
       *  Switch: '<S423>/Switch5'
       */
      if (1.0 >= fabs(rtb_Sum1_dh)) {
        rtb_Switch_n = 1.0;
      } else {
        rtb_Switch_n = rtb_Sum1_dh;
      }

      /* End of Switch: '<S449>/Switch' */

      /* Sum: '<S423>/Sum5' incorporates:
       *  Switch: '<S423>/Switch5'
       */
      rtb_Sum1_dh = Gen2_ref_B->BusInput3.leanox.rP_1 +
        Gen2_ref_B->BusInput3.leanox.rP_Eng_Frict;

      /* Switch: '<S457>/Switch' incorporates:
       *  Abs: '<S457>/Abs'
       *  Constant: '<S457>/Constant2'
       *  RelationalOperator: '<S457>/Relational Operator'
       *  Switch: '<S423>/Switch5'
       */
      if (1.0 >= fabs(Gen2_ref_B->BusInput3.leanox.rT_1)) {
        rtb_bResetHlci_0 = 1.0;
      } else {
        rtb_bResetHlci_0 = Gen2_ref_B->BusInput3.leanox.rT_1;
      }

      /* End of Switch: '<S457>/Switch' */

      /* Switch: '<S448>/Switch' incorporates:
       *  Abs: '<S448>/Abs'
       *  Constant: '<S448>/Constant2'
       *  RelationalOperator: '<S448>/Relational Operator'
       *  Switch: '<S423>/Switch5'
       */
      if (1.0 >= fabs(rtb_Sum1_dh)) {
        rtb_Sum1_dh = 1.0;
      }

      /* End of Switch: '<S448>/Switch' */

      /* Product: '<S423>/rKK3' incorporates:
       *  Switch: '<S423>/Switch5'
       */
      rtb_Sum1_dh = Gen2_ref_B->BusInput3.leanox.rPr_mbar_1 *
        Gen2_ref_B->BusInput3.leanox.rN_1 / rtb_bResetHlci_0 / rtb_Sum1_dh;

      /* Switch: '<S450>/Switch' incorporates:
       *  Abs: '<S450>/Abs'
       *  Constant: '<S450>/Constant2'
       *  RelationalOperator: '<S450>/Relational Operator'
       *  Switch: '<S423>/Switch5'
       */
      if (1.0 >= fabs(Gen2_ref_B->BusInput3.leanox.rT_c)) {
        rtb_bResetHlci_0 = 1.0;
      } else {
        rtb_bResetHlci_0 = Gen2_ref_B->BusInput3.leanox.rT_c;
      }

      /* End of Switch: '<S450>/Switch' */

      /* Switch: '<S458>/Switch' incorporates:
       *  Abs: '<S458>/Abs'
       *  Constant: '<S458>/Constant2'
       *  RelationalOperator: '<S458>/Relational Operator'
       *  Switch: '<S423>/Switch5'
       */
      if (1.0 >= fabs(rtb_Product4_d)) {
        rtb_Product4_d = 1.0;
      }

      /* End of Switch: '<S458>/Switch' */

      /* Switch: '<S423>/Switch5' incorporates:
       *  Product: '<S423>/Divide10'
       *  Product: '<S423>/Divide9'
       *  Product: '<S423>/rKK4'
       *  Sum: '<S423>/Add3'
       *  Sum: '<S423>/Sum6'
       *  Sum: '<S423>/Sum7'
       */
      rtb_Sum4_ny = (rtb_Sum1_dh - Gen2_ref_B->BusInput3.leanox.rPr_mbar_c *
                     Gen2_ref_B->BusInput3.leanox.rN_c / rtb_bResetHlci_0 /
                     rtb_Switch_n) / rtb_Product4_d * (rtb_Sum4_ny -
        Gen2_ref_B->BusInput3.leanox.rP_1) + rtb_Sum1_dh;
    } else {
      /* Sum: '<S423>/Add10' incorporates:
       *  Switch: '<S423>/Switch5'
       */
      rtb_Product4_d = Gen2_ref_B->BusInput3.leanox.rP_2 -
        Gen2_ref_B->BusInput3.leanox.rP_1;

      /* Sum: '<S423>/Sum' incorporates:
       *  Switch: '<S423>/Switch5'
       */
      rtb_Switch_n = Gen2_ref_B->BusInput3.leanox.rP_1 +
        Gen2_ref_B->BusInput3.leanox.rP_Eng_Frict;

      /* Sum: '<S423>/Sum1' incorporates:
       *  Switch: '<S423>/Switch5'
       */
      rtb_Sum1_dh = Gen2_ref_B->BusInput3.leanox.rP_2 +
        Gen2_ref_B->BusInput3.leanox.rP_Eng_Frict;

      /* Switch: '<S447>/Switch' incorporates:
       *  Abs: '<S447>/Abs'
       *  Constant: '<S447>/Constant2'
       *  RelationalOperator: '<S447>/Relational Operator'
       *  Switch: '<S423>/Switch5'
       */
      if (1.0 >= fabs(Gen2_ref_B->BusInput3.leanox.rT_2)) {
        rtb_bResetHlci_0 = 1.0;
      } else {
        rtb_bResetHlci_0 = Gen2_ref_B->BusInput3.leanox.rT_2;
      }

      /* End of Switch: '<S447>/Switch' */

      /* Switch: '<S452>/Switch' incorporates:
       *  Abs: '<S452>/Abs'
       *  Constant: '<S452>/Constant2'
       *  RelationalOperator: '<S452>/Relational Operator'
       *  Switch: '<S423>/Switch5'
       */
      if (1.0 >= fabs(rtb_Sum1_dh)) {
        rtb_Sum1_dh = 1.0;
      }

      /* End of Switch: '<S452>/Switch' */

      /* Product: '<S423>/rKK1' incorporates:
       *  Switch: '<S423>/Switch5'
       */
      rtb_Sum1_dh = Gen2_ref_B->BusInput3.leanox.rPr_mbar_2 *
        Gen2_ref_B->BusInput3.leanox.rN_2 / rtb_bResetHlci_0 / rtb_Sum1_dh;

      /* Switch: '<S453>/Switch' incorporates:
       *  Abs: '<S453>/Abs'
       *  Constant: '<S453>/Constant2'
       *  RelationalOperator: '<S453>/Relational Operator'
       *  Switch: '<S423>/Switch5'
       */
      if (1.0 >= fabs(rtb_Switch_n)) {
        rtb_Switch_n = 1.0;
      }

      /* End of Switch: '<S453>/Switch' */

      /* Switch: '<S451>/Switch' incorporates:
       *  Abs: '<S451>/Abs'
       *  Constant: '<S451>/Constant2'
       *  RelationalOperator: '<S451>/Relational Operator'
       *  Switch: '<S423>/Switch5'
       */
      if (1.0 >= fabs(rtb_Product4_d)) {
        rtb_Product4_d = 1.0;
      }

      /* End of Switch: '<S451>/Switch' */

      /* Switch: '<S423>/Switch5' incorporates:
       *  Product: '<S423>/Divide2'
       *  Product: '<S423>/Divide3'
       *  Product: '<S423>/rKK2'
       *  Sum: '<S423>/Add2'
       *  Sum: '<S423>/Sum2'
       *  Sum: '<S423>/Sum3'
       */
      rtb_Sum4_ny = (rtb_Sum1_dh - Gen2_ref_B->BusInput3.leanox.rPr_mbar_1 *
                     Gen2_ref_B->BusInput3.leanox.rN_1 /
                     Gen2_ref_B->BusInput3.leanox.rT_1 / rtb_Switch_n) /
        rtb_Product4_d * (rtb_Sum4_ny - Gen2_ref_B->BusInput3.leanox.rP_2) +
        rtb_Sum1_dh;
    }

    rtb_Product4_d = rtb_Sum4_ny * Gen2_ref_B->T2s_filt.Switch *
      (Gen2_ref_B->BusInput3.leanox.rP_Eng_Frict + rtb_Switch2_jq) /
      rtb_MinMax_a;
  }

  /* End of Switch: '<S423>/Switch2' */

  /* Product: '<S459>/Divide8' incorporates:
   *  DataTypeConversion: '<S459>/Data Type Conversion2'
   */
  rtb_Sum4_ny = rtb_Product4_d * Gen2_ref_B->BusInput.tLEANOXin.rLEANOX_fact_BC;

  /* MinMax: '<S459>/MinMax' */
  rtb_Product4_d = rtb_Divide5_h;

  /* Product: '<S459>/Divide5' incorporates:
   *  Delay: '<S15>/Resettable Delay'
   *  Sum: '<S459>/Add9'
   */
  rtb_Divide5_h = ((rtb_Sum_c + rtb_Sum4_ny) +
                   Gen2_ref_DWork->ResettableDelay_DSTATE) * rtb_Product4_d;

  /* DataTypeConversion: '<S459>/Data Type Conversion' */
  rtb_Product4_d = Gen2_ref_B->BusInput.tLEANOXin.rLEANOXoffset;

  /* Gain: '<S459>/mbar2pa' incorporates:
   *  Sum: '<S459>/Add1'
   */
  rtb_mbar2pa_i = (rtb_Divide5_h + rtb_Product4_d) * 100.0;

  /* Sum: '<S430>/Sum2' incorporates:
   *  Gain: '<S430>/pa2mbar'
   *  Product: '<S8>/Product3'
   */
  rtb_Divide2_f = rtb_Divide2_f * rtb_mbar2pa_i * 0.01 +
    Gen2_ref_B->BusInput3.leanox.rPr_Offset_Island;

  /* Switch: '<S624>/Switch2' incorporates:
   *  RelationalOperator: '<S624>/LowerRelop1'
   */
  if (!(rtb_Divide2_f > r)) {
    /* Gain: '<S430>/bar2mbar2' */
    rtb_Divide5_h = 1000.0 * Gen2_ref_B->BusInput3.traj.rPr_p2s_min;

    /* Switch: '<S624>/Switch' incorporates:
     *  RelationalOperator: '<S624>/UpperRelop'
     */
    if (rtb_Divide2_f < rtb_Divide5_h) {
      r = rtb_Divide5_h;
    } else {
      r = rtb_Divide2_f;
    }

    /* End of Switch: '<S624>/Switch' */
  }

  /* End of Switch: '<S624>/Switch2' */

  /* Outputs for Atomic SubSystem: '<S8>/Filter' */
  /* Gain: '<S430>/mbar2pa1' */
  Gen2_ref_Pd_filt(100.0 * r, Gen2_ref_B->BusInput3.SpeedCtrl.rTi_p2s_LEANOX,
                   rtb_Switch_i5[5], rtb_bResetHlci, &Gen2_ref_B->Filter_k,
                   &Gen2_ref_DWork->Filter_k, inst);

  /* End of Outputs for SubSystem: '<S8>/Filter' */

  /* Switch: '<Root>/BDC_traj4' */
  if (rtb_LogicalOperator) {
    r = rtb_Pa2bar_k;
  } else {
    r = Gen2_ref_B->Filter_k.Switch;
  }

  /* End of Switch: '<Root>/BDC_traj4' */

  /* Gain: '<S16>/Pa2bar1' */
  rtb_Sum_e = 1.0E-5 * r;

  /* Gain: '<S889>/Gain' */
  r = 0.001 * Gen2_ref_B->Pel_filt.Switch;

  /* Sum: '<S889>/Sum' */
  rtb_Divide2_f = Gen2_ref_B->BusInput3.SkipF.rNum_max_P1 -
    Gen2_ref_B->BusInput3.SkipF.rNum_max_P0;

  /* Sum: '<S889>/Sum1' */
  rtb_Product4_d = Gen2_ref_B->BusInput3.SkipF.rP_max_1 -
    Gen2_ref_B->BusInput3.SkipF.rP_max_0;

  /* Switch: '<S904>/Switch' incorporates:
   *  Abs: '<S904>/Abs'
   *  Constant: '<S904>/Constant2'
   *  RelationalOperator: '<S904>/Relational Operator'
   */
  if (2.2204460492503131E-16 >= fabs(rtb_Product4_d)) {
    rtb_Product4_d = 2.2204460492503131E-16;
  }

  /* End of Switch: '<S904>/Switch' */

  /* Sum: '<S889>/Sum3' incorporates:
   *  Product: '<S889>/Divide'
   *  Sum: '<S889>/Sum2'
   */
  rtb_Divide2_f = (r - Gen2_ref_B->BusInput3.SkipF.rP_max_0) * rtb_Divide2_f /
    rtb_Product4_d + Gen2_ref_B->BusInput3.SkipF.rNum_max_P0;

  /* Switch: '<S905>/Switch2' incorporates:
   *  Constant: '<S889>/Constant5'
   *  RelationalOperator: '<S905>/LowerRelop1'
   *  RelationalOperator: '<S905>/UpperRelop'
   *  Switch: '<S905>/Switch'
   */
  if (rtb_Divide2_f > Gen2_ref_B->BusInput3.SkipF.rNum_max) {
    r = Gen2_ref_B->BusInput3.SkipF.rNum_max;
  } else if (rtb_Divide2_f < 0.0) {
    /* Switch: '<S905>/Switch' incorporates:
     *  Constant: '<S889>/Constant5'
     */
    r = 0.0;
  } else {
    r = rtb_Divide2_f;
  }

  /* End of Switch: '<S905>/Switch2' */

  /* Rounding: '<S889>/Rounding Function' */
  rtb_RoundingFunction = rt_roundd_snf(r, inst);

  /* Gain: '<S427>/Gain9' incorporates:
   *  Gain: '<S427>/Gain10'
   *  Gain: '<S427>/Gain11'
   */
  r = 0.001 * Gen2_ref_B->BusInput3.LR.iTime_Eng_Cyc;

  /* Bias: '<S427>/ u+Ts1' incorporates:
   *  Product: '<S427>/Product1'
   */
  rtb_Divide2_f = r * Gen2_ref_B->BusInput3.LR.iCyc_Ign_Max_Off + 0.01;

  /* Outputs for Atomic SubSystem: '<S427>/TP_Misfire_ON' */
  /* Logic: '<S427>/Logical Operator3' incorporates:
   *  Delay: '<S427>/Delay'
   *  Logic: '<S427>/Logical Operator24'
   *  RelationalOperator: '<S427>/Relational Operator1'
   *  RelationalOperator: '<S427>/Relational Operator6'
   *  UnitDelay: '<S427>/Unit Delay5'
   */
  Gen2_ref_TP_ActSat_CBV(((!Gen2_ref_DWork->TOF_2_state) &&
    rtb_RelationalOperator2_j && (Gen2_ref_DWork->Delay_DSTATE[0] >=
    Gen2_ref_B->BusInput3.LR.rP_LR_Trig_Misf) && (rtb_Saturation >
    Gen2_ref_B->BusInput3.LR.rP_LR_Trig_Misf) &&
    Gen2_ref_B->BusInput3.LR.bP_LoadReject_Active), rtb_Divide2_f,
    &Gen2_ref_B->TP_Misfire_ON, &Gen2_ref_DWork->TP_Misfire_ON, inst);

  /* End of Outputs for SubSystem: '<S427>/TP_Misfire_ON' */

  /* Bias: '<S427>/ u+Ts8' incorporates:
   *  Product: '<S427>/Product2'
   */
  rtb_Divide5_h = r * Gen2_ref_B->BusInput3.LR.iCyc_Ign_Min_On + 0.01;

  /* Outputs for Atomic SubSystem: '<S427>/TP_Misfire_OFF' */
  /* Logic: '<S427>/Logical Operator6' */
  Gen2_ref_TP_ActSat_CBV(!Gen2_ref_B->TP_Misfire_ON.LogicalOperator1,
    rtb_Divide5_h, &Gen2_ref_B->TP_Misfire_OFF, &Gen2_ref_DWork->TP_Misfire_OFF, inst);

  /* End of Outputs for SubSystem: '<S427>/TP_Misfire_OFF' */

  /* Logic: '<S427>/Logical Operator8' incorporates:
   *  Logic: '<S427>/Logical Operator18'
   *  Switch: '<S427>/Switch'
   */
  rtb_bCBV_min = !Gen2_ref_B->TP_Misfire_OFF.LogicalOperator1;

  /* Outputs for Atomic SubSystem: '<S427>/TP_Misfire_OFF1' */
  /* Sum: '<S427>/Sum' incorporates:
   *  Gain: '<S427>/Gain12'
   */
  Gen2_ref_TP_ActSat_CBV(Gen2_ref_B->TP_Misfire_ON.LogicalOperator1, 2.0 *
    rtb_Divide2_f + rtb_Divide5_h, &Gen2_ref_B->TP_Misfire_OFF1,
    &Gen2_ref_DWork->TP_Misfire_OFF1, inst);

  /* End of Outputs for SubSystem: '<S427>/TP_Misfire_OFF1' */

  /* Switch: '<S427>/Switch2' incorporates:
   *  Constant: '<S427>/Constant1'
   *  Logic: '<S427>/Logical Operator19'
   *  Logic: '<S427>/Logical Operator5'
   *  UnitDelay: '<S427>/Unit Delay2'
   *  UnitDelay: '<S427>/Unit Delay3'
   */
  if (Gen2_ref_B->TP_Misfire_ON.LogicalOperator1) {
    rtb_dbg_HLCi = true;
  } else {
    rtb_dbg_HLCi = (Gen2_ref_B->TP_Misfire_OFF1.LogicalOperator1 &&
                    (!Gen2_ref_DWork->UnitDelay3_DSTATE_h5) &&
                    Gen2_ref_DWork->UnitDelay2_DSTATE_hh);
  }

  /* End of Switch: '<S427>/Switch2' */

  /* Switch: '<S427>/Switch' incorporates:
   *  Constant: '<S427>/Constant4'
   *  DataTypeConversion: '<S4>/Data Type Conversion34'
   *  Logic: '<S427>/Logical Operator20'
   *  Logic: '<S427>/Logical Operator21'
   *  RelationalOperator: '<S427>/Relational Operator9'
   *  Switch: '<S427>/Switch3'
   */
  if (Gen2_ref_B->BusInput.rN_Eng_LRskipF >
      Gen2_ref_B->BusInput3.LR.rN_Misf_2_Trig) {
    rtb_LogicalOperator2_ov = (rtb_bCBV_min &&
      (!Gen2_ref_B->TP_Misfire_ON.LogicalOperator1) && rtb_dbg_HLCi);
  } else {
    rtb_LogicalOperator2_ov = false;
  }

  /* Outputs for Atomic SubSystem: '<S427>/TP_Misfire_ON_2nd time' */
  /* Bias: '<S427>/ u+Ts9' incorporates:
   *  Product: '<S427>/Product3'
   */
  Gen2_ref_TP_ActSat_CBV(rtb_LogicalOperator2_ov, r *
    Gen2_ref_B->BusInput3.LR.iCyc_Ign_Max_Off + 0.01,
    &Gen2_ref_B->TP_Misfire_ON_2ndtime, &Gen2_ref_DWork->TP_Misfire_ON_2ndtime, inst);

  /* End of Outputs for SubSystem: '<S427>/TP_Misfire_ON_2nd time' */

  /* Outputs for Atomic SubSystem: '<S427>/TP_Misfire_OFF2' */
  /* Logic: '<S427>/Logical Operator22' */
  Gen2_ref_TP_ActSat_CBV(!Gen2_ref_B->TP_Misfire_ON_2ndtime.LogicalOperator1,
    rtb_Divide5_h, &Gen2_ref_B->TP_Misfire_OFF2,
    &Gen2_ref_DWork->TP_Misfire_OFF2, inst);

  /* End of Outputs for SubSystem: '<S427>/TP_Misfire_OFF2' */

  /* Logic: '<S427>/Logical Operator23' */
  rtb_bTV_sat = !Gen2_ref_B->TP_Misfire_OFF2.LogicalOperator1;

  /* Logic: '<S427>/Logical Operator9' incorporates:
   *  Logic: '<S427>/Logical Operator10'
   *  Logic: '<S427>/Logical Operator7'
   *  Logic: '<S427>/Logical Operator8'
   */
  rtb_bCBV_min = ((Gen2_ref_B->TP_Misfire_ON.LogicalOperator1 && rtb_bCBV_min &&
                   rtb_bTV_sat) || (rtb_bCBV_min &&
    Gen2_ref_B->TP_Misfire_ON_2ndtime.LogicalOperator1 && rtb_bTV_sat));

  /* Switch: '<S19>/Switch2' incorporates:
   *  Constant: '<S19>/Constant2'
   */
  if (rtb_bCBV_min) {
    rtb_Switch2_d1 = rtb_RoundingFunction;
  } else {
    rtb_Switch2_d1 = 0.0;
  }

  /* End of Switch: '<S19>/Switch2' */

  /* Gain: '<S896>/Gain5' incorporates:
   *  DataTypeConversion: '<S4>/Data Type Conversion16'
   *  Sum: '<S19>/Sum'
   */
  rtb_Divide2_f = -(Gen2_ref_B->BusInput.rN_Set - rtb_DataTypeConversion15);

  /* Switch: '<S907>/Switch2' incorporates:
   *  Constant: '<S896>/  1'
   *  RelationalOperator: '<S907>/LowerRelop1'
   *  RelationalOperator: '<S907>/UpperRelop'
   *  Switch: '<S907>/Switch'
   */
  if (rtb_Divide2_f > 500.0) {
    r = 500.0;
  } else if (rtb_Divide2_f < Gen2_ref_B->BusInput3.SkipF.rN_Active_Lim) {
    /* Switch: '<S907>/Switch' */
    r = Gen2_ref_B->BusInput3.SkipF.rN_Active_Lim;
  } else {
    r = rtb_Divide2_f;
  }

  /* End of Switch: '<S907>/Switch2' */

  /* Product: '<S896>/Product1' incorporates:
   *  Sum: '<S896>/Sum3'
   */
  rtb_Product1_mqz = (r - Gen2_ref_B->BusInput3.SkipF.rN_Active_Lim) *
    Gen2_ref_B->BusInput3.SkipF.rKp;

  /* Outputs for Atomic SubSystem: '<S19>/Filter' */
  Gen2_ref_Filter3(rtb_Product1_mqz, Gen2_ref_B->BusInput3.SkipF.rTiF_Num,
                   Gen2_ref_ConstB.x0_f, rtb_bResetBdc, &Gen2_ref_B->Filter_mn,
                   &Gen2_ref_DWork->Filter_mn, inst);

  /* End of Outputs for SubSystem: '<S19>/Filter' */

  /* Switch: '<S19>/Switch1' incorporates:
   *  Constant: '<S19>/  1'
   *  Logic: '<S19>/Logical Operator'
   */
  if (Gen2_ref_B->BusInput3.eng.bPI_engine ||
      Gen2_ref_B->BusInput3.eng.bActive_MisfCtrl) {
    /* Switch: '<S893>/Switch2' incorporates:
     *  Constant: '<S19>/Constant23'
     *  RelationalOperator: '<S893>/LowerRelop1'
     *  RelationalOperator: '<S893>/UpperRelop'
     *  Switch: '<S893>/Switch'
     */
    if (Gen2_ref_B->Filter_mn.Switch > rtb_RoundingFunction) {
      rtb_Divide2_f = rtb_RoundingFunction;
    } else if (Gen2_ref_B->Filter_mn.Switch < 0.0) {
      /* Switch: '<S893>/Switch' incorporates:
       *  Constant: '<S19>/Constant23'
       */
      rtb_Divide2_f = 0.0;
    } else {
      rtb_Divide2_f = Gen2_ref_B->Filter_mn.Switch;
    }

    /* End of Switch: '<S893>/Switch2' */
  } else {
    rtb_Divide2_f = 0.0;
  }

  /* End of Switch: '<S19>/Switch1' */

  /* MATLAB Function: '<S19>/MATLAB Function' */
  Gen2_ref_MATLABFunction_n(rtb_Divide2_f, Gen2_ref_B->BusInput3.SkipF.rHy_eps,
    &Gen2_ref_B->sf_MATLABFunction_i, &Gen2_ref_DWork->sf_MATLABFunction_i, inst);

  /* MATLAB Function: '<S633>/MATLAB Function' */
  Gen2_ref_MATLABFunction_n(rtb_Product_m[3],
    Gen2_ref_B->BusInput3.SkipF.rHy_eps, &Gen2_ref_B->sf_MATLABFunction_kd,
    &Gen2_ref_DWork->sf_MATLABFunction_kd, inst);

  /* Switch: '<S19>/NSkip' incorporates:
   *  Switch: '<S8>/Switch1'
   */
  if (rtb_LogicalOperator) {
    rtb_Divide2_f = rtb_MinMax_n;
  } else {
    if (Gen2_ref_B->BusInput3.SkipF.bSF_ON) {
      /* Switch: '<S8>/Switch9' incorporates:
       *  DataTypeConversion: '<S8>/Data Type Conversion2'
       *  Logic: '<S8>/Logical Operator1'
       *  Product: '<S8>/Product2'
       *  Sum: '<S429>/Sum9'
       *  Switch: '<S8>/Switch1'
       */
      if (!Gen2_ref_B->BusInput3.SpeedCtrl.bSF_OFF_iLQR) {
        rtb_Divide2_f = Gen2_ref_B->sf_MATLABFunction_kd.y;
      } else {
        rtb_Divide2_f = (rtb_Switch2_ba + rtb_Switch5_iq) * (real_T)
          Gen2_ref_B->BusInput3.SkipF.bSF_ON;
      }

      /* End of Switch: '<S8>/Switch9' */
    } else {
      /* Switch: '<S8>/Switch1' incorporates:
       *  Constant: '<S8>/Constant3'
       */
      rtb_Divide2_f = 0.0;
    }

    /* Sum: '<S19>/Sum1' incorporates:
     *  Switch: '<S19>/Switch4'
     */
    rtb_Divide2_f += rtb_Switch2_d1;

    /* Switch: '<S895>/Switch2' incorporates:
     *  Constant: '<S19>/Constant4'
     *  RelationalOperator: '<S895>/LowerRelop1'
     *  RelationalOperator: '<S895>/UpperRelop'
     *  Switch: '<S895>/Switch'
     */
    if (rtb_Divide2_f > rtb_RoundingFunction) {
      rtb_Divide2_f = rtb_RoundingFunction;
    } else if (rtb_Divide2_f < 0.0) {
      /* Switch: '<S895>/Switch' incorporates:
       *  Constant: '<S19>/Constant4'
       */
      rtb_Divide2_f = 0.0;
    }

    /* End of Switch: '<S895>/Switch2' */
  }

  /* End of Switch: '<S19>/NSkip' */

  /* Switch: '<S894>/Switch2' incorporates:
   *  Constant: '<S19>/Constant3'
   *  RelationalOperator: '<S894>/LowerRelop1'
   *  RelationalOperator: '<S894>/UpperRelop'
   *  Switch: '<S894>/Switch'
   */
  if (rtb_Divide2_f > Gen2_ref_B->BusInput3.eng.rNum_Cyl_Eng) {
    r = Gen2_ref_B->BusInput3.eng.rNum_Cyl_Eng;
  } else if (rtb_Divide2_f < 0.0) {
    /* Switch: '<S894>/Switch' incorporates:
     *  Constant: '<S19>/Constant3'
     */
    r = 0.0;
  } else {
    r = rtb_Divide2_f;
  }

  /* End of Switch: '<S894>/Switch2' */

  /* DataTypeConversion: '<S16>/Data Type Conversion9' */
  rtb_bResetHlci_0 = floor(r);
  if (rtIsNaN(rtb_bResetHlci_0) || rtIsInf(rtb_bResetHlci_0)) {
    rtb_bResetHlci_0 = 0.0;
  } else {
    rtb_bResetHlci_0 = fmod(rtb_bResetHlci_0, 65536.0);
  }

  /* BusCreator: '<S16>/Bus Creator' incorporates:
   *  DataTypeConversion: '<S16>/Data Type Conversion9'
   *  Outport: '<Root>/out'
   */
  Gen2_ref_Y->out.iNskip = (int16_T)(rtb_bResetHlci_0 < 0.0 ? (int32_T)(int16_T)
    -(int16_T)(uint16_T)-rtb_bResetHlci_0 : (int32_T)(int16_T)(uint16_T)
    rtb_bResetHlci_0);

  /* Abs: '<S9>/Abs1' */
  rtb_Divide2_f = fabs(Gen2_ref_B->BusInput3.ITC.rITCdeltaMAX);

  /* S-Function (sfix_look1_dyn): '<S634>/Lookup Table Dynamic1' */
  /* Dynamic Look-Up Table Block: '<S634>/Lookup Table Dynamic1'
   * Input0  Data Type:  Floating Point real_T
   * Input1  Data Type:  Floating Point real_T
   * Input2  Data Type:  Floating Point real_T
   * Output0 Data Type:  Floating Point real_T
   * Lookup Method: Linear_Endpoint
   *
   */
  LookUp_real_T_real_T( &(rtb_LookupTableDynamic1),
                       &Gen2_ref_B->BusInput3.ITC.rITCtransDeltaAcc_y[0],
                       rtb_Gain3, &Gen2_ref_B->
                       BusInput3.ITC.rITCtransDeltaAcc_x[0], 4U, inst);

  /* Abs: '<S634>/Abs2' incorporates:
   *  Abs: '<S9>/Abs4'
   */
  rtb_Sum4_ny = fabs(Gen2_ref_B->BusInput3.ITC.rITCtransSRback);

  /* Product: '<S708>/delta rise limit' incorporates:
   *  Abs: '<S634>/Abs2'
   *  Gain: '<S634>/Gain2'
   *  Product: '<S811>/delta rise limit'
   *  SampleTimeMath: '<S708>/sample time'
   *
   * About '<S708>/sample time':
   *  y = K where K = ( w * Ts )
   */
  x = 1000.0 * rtb_Sum4_ny * 0.01;
  rtb_Product4_d = x;

  /* Switch: '<S634>/Switch' incorporates:
   *  RelationalOperator: '<S634>/Relational Operator2'
   *  UnitDelay: '<S634>/Unit Delay'
   */
  rtb_bTriger_IT_LJ = ((delta_y_tmp_tmp >
                        Gen2_ref_B->BusInput3.ITC.rITCtransDPthrsh) ||
                       Gen2_ref_DWork->UnitDelay_DSTATE_kx);

  /* Outputs for Atomic SubSystem: '<S634>/Delay Retard' */
  Gen2_ref_TON_1(rtb_bTriger_IT_LJ, Gen2_ref_B->BusInput3.ITC.rITCtransDelay,
                 &Gen2_ref_B->DelayRetard, &Gen2_ref_DWork->DelayRetard, inst);

  /* End of Outputs for SubSystem: '<S634>/Delay Retard' */

  /* Switch: '<S634>/Switch1' incorporates:
   *  Abs: '<S634>/Abs1'
   *  Constant: '<S634>/Constant7'
   */
  if (Gen2_ref_B->DelayRetard.LogicalOperator3) {
    rtb_Sum_c = fabs(rtb_LookupTableDynamic1);
  } else {
    rtb_Sum_c = 0.0;
  }

  /* End of Switch: '<S634>/Switch1' */

  /* Delay: '<S708>/Delay' incorporates:
   *  Constant: '<S634>/Constant3'
   *  Delay: '<S425>/Delay'
   */
  Gen2_ref_DWork->icLoad_nv = ((((Gen2_ref_PrevZCSigState->Delay_Reset_ZCE_j ==
    1) != (int32_T)rtb_bResetHlci) &&
    (Gen2_ref_PrevZCSigState->Delay_Reset_ZCE_j != 3)) || rtb_bResetHlci ||
    Gen2_ref_DWork->icLoad_nv);
  Gen2_ref_PrevZCSigState->Delay_Reset_ZCE_j = rtb_bResetHlci;
  if (Gen2_ref_DWork->icLoad_nv) {
    Gen2_ref_DWork->Delay_DSTATE_l = 0.0;
  }

  /* Switch: '<S708>/etaVolConst' incorporates:
   *  Constant: '<S634>/Constant3'
   */
  if (rtb_bResetHlci) {
    rtb_bResetHlci_0 = 0.0;
  } else {
    rtb_bResetHlci_0 = rtb_Sum_c;
  }

  /* End of Switch: '<S708>/etaVolConst' */

  /* Sum: '<S708>/Difference Inputs1' incorporates:
   *  Delay: '<S708>/Delay'
   */
  rtb_Divide5_h = rtb_bResetHlci_0 - Gen2_ref_DWork->Delay_DSTATE_l;

  /* Switch: '<S711>/Switch2' incorporates:
   *  RelationalOperator: '<S711>/LowerRelop1'
   */
  if (!(rtb_Divide5_h > rtb_Product4_d)) {
    /* Product: '<S708>/delta fall limit' incorporates:
     *  Abs: '<S634>/Abs2'
     *  Gain: '<S634>/Gain1'
     *  SampleTimeMath: '<S708>/sample time'
     *
     * About '<S708>/sample time':
     *  y = K where K = ( w * Ts )
     */
    rtb_Switch5_iq = -rtb_Sum4_ny * 0.01;

    /* Switch: '<S711>/Switch' incorporates:
     *  RelationalOperator: '<S711>/UpperRelop'
     */
    if (rtb_Divide5_h < rtb_Switch5_iq) {
      rtb_Product4_d = rtb_Switch5_iq;
    } else {
      rtb_Product4_d = rtb_Divide5_h;
    }

    /* End of Switch: '<S711>/Switch' */
  }

  /* End of Switch: '<S711>/Switch2' */

  /* Sum: '<S708>/Difference Inputs2' incorporates:
   *  Delay: '<S708>/Delay'
   */
  rtb_Divide5_h = rtb_Product4_d + Gen2_ref_DWork->Delay_DSTATE_l;

  /* Signum: '<S634>/Sign' */
  if (rtb_LookupTableDynamic1 < 0.0) {
    rtb_bResetHlci_0 = -1.0;
  } else if (rtb_LookupTableDynamic1 > 0.0) {
    rtb_bResetHlci_0 = 1.0;
  } else if (rtb_LookupTableDynamic1 == 0.0) {
    rtb_bResetHlci_0 = 0.0;
  } else {
    rtb_bResetHlci_0 = (rtNaN);
  }

  /* End of Signum: '<S634>/Sign' */

  /* MinMax: '<S634>/MinMax' */
  if ((rtb_Divide5_h >= rtb_Sum_c) || rtIsNaN(rtb_Sum_c)) {
    rtb_Sum_c = rtb_Divide5_h;
  }

  /* End of MinMax: '<S634>/MinMax' */

  /* Product: '<S634>/Product' */
  rtb_Product4_d = rtb_bResetHlci_0 * rtb_Sum_c;

  /* Sum: '<S431>/Sum' */
  rtb_Sum_c = rtb_Product_m[2] + rtb_Product4_d;

  /* Gain: '<S427>/Gain8' */
  rtb_Sum1_dh = 1000.0 * Gen2_ref_B->BusInput3.LR.rRateITadvance;

  /* Product: '<S524>/delta rise limit' incorporates:
   *  SampleTimeMath: '<S524>/sample time'
   *
   * About '<S524>/sample time':
   *  y = K where K = ( w * Ts )
   */
  rtb_Sum1_dh *= 0.01;

  /* Outputs for Atomic SubSystem: '<S427>/TP_Ign retard' */
  /* Logic: '<S427>/Logical Operator4' incorporates:
   *  Bias: '<S427>/ u+Ts2'
   *  Gain: '<S427>/Gain13'
   *  RelationalOperator: '<S427>/Relational Operator2'
   */
  Gen2_ref_TP_ActSat_CBV(((rtb_Saturation >
    Gen2_ref_B->BusInput3.LR.rP_LR_Trig_IGN_Retard) &&
    Gen2_ref_B->BusInput3.LR.bP_LoadReject_Active && rtb_RelationalOperator2_j),
    0.001 * Gen2_ref_B->BusInput3.LR.rTi_LR_IGN_Retard_MAX + 0.01,
    &Gen2_ref_B->TP_Ignretard, &Gen2_ref_DWork->TP_Ignretard, inst);

  /* End of Outputs for SubSystem: '<S427>/TP_Ign retard' */

  /* Logic: '<S427>/Logical Operator12' incorporates:
   *  Logic: '<S427>/Logical Operator13'
   *  RelationalOperator: '<S427>/Relational Operator4'
   *  UnitDelay: '<S427>/Unit Delay'
   */
  rtb_RelationalOperator2_j = (rtb_TOF_IN ||
    Gen2_ref_B->TP_Ignretard.LogicalOperator1 || ((rtb_Divide4_d >
    Gen2_ref_B->BusInput3.LR.rN_LR_IGN_Retard_ON) &&
    Gen2_ref_DWork->UnitDelay_DSTATE_n));

  /* Sum: '<S427>/Sum2' */
  rtb_MinMax_a = Gen2_ref_B->BusInput3.LR.rProt_IGN_Retard_max -
    Gen2_ref_B->BusInput3.LR.rProt_IGN_Retard_min;

  /* Abs: '<S506>/Abs' */
  rtb_Switch_n = fabs(rtb_MinMax_a);

  /* Switch: '<S506>/Switch' incorporates:
   *  Constant: '<S506>/Constant2'
   *  RelationalOperator: '<S506>/Relational Operator'
   */
  if (2.2204460492503131E-16 >= rtb_Switch_n) {
    rtb_MinMax_a = 2.2204460492503131E-16;
  }

  /* End of Switch: '<S506>/Switch' */

  /* Sum: '<S427>/Sum4' incorporates:
   *  Product: '<S427>/Divide'
   *  Product: '<S427>/Product'
   *  Sum: '<S427>/Sum1'
   *  Sum: '<S427>/Sum3'
   */
  rtb_Divide4_d = (rtb_Saturation -
                   Gen2_ref_B->BusInput3.LR.rProt_IGN_Retard_min) / rtb_MinMax_a
    * (Gen2_ref_B->BusInput3.LR.rLR_IGN_Retard_IT -
       Gen2_ref_B->BusInput3.LR.rLR_IGN_Retard_IT_min) +
    Gen2_ref_B->BusInput3.LR.rLR_IGN_Retard_IT_min;

  /* Switch: '<S510>/Switch2' incorporates:
   *  RelationalOperator: '<S510>/LowerRelop1'
   *  RelationalOperator: '<S510>/UpperRelop'
   *  Switch: '<S510>/Switch'
   */
  if (rtb_Divide4_d > Gen2_ref_B->BusInput3.LR.rLR_IGN_Retard_IT) {
    rtb_Switch2_jq = Gen2_ref_B->BusInput3.LR.rLR_IGN_Retard_IT;
  } else if (rtb_Divide4_d < Gen2_ref_B->BusInput3.LR.rLR_IGN_Retard_IT_min) {
    /* Switch: '<S510>/Switch' */
    rtb_Switch2_jq = Gen2_ref_B->BusInput3.LR.rLR_IGN_Retard_IT_min;
  } else {
    rtb_Switch2_jq = rtb_Divide4_d;
  }

  /* End of Switch: '<S510>/Switch2' */

  /* Switch: '<S427>/Switch6' incorporates:
   *  UnitDelay: '<S427>/Unit Delay6'
   */
  if (rtb_RelationalOperator2_j) {
    rtb_MinMax_a = Gen2_ref_DWork->UnitDelay6_DSTATE_m;
  } else {
    rtb_MinMax_a = rtb_Switch2_jq;
  }

  /* End of Switch: '<S427>/Switch6' */

  /* MinMax: '<S427>/MinMax1' */
  if ((rtb_MinMax_a >= rtb_Switch2_jq) || rtIsNaN(rtb_Switch2_jq)) {
    rtb_Divide4_d = rtb_MinMax_a;
  } else {
    rtb_Divide4_d = rtb_Switch2_jq;
  }

  /* End of MinMax: '<S427>/MinMax1' */

  /* Switch: '<S427>/Ign retard type 6' incorporates:
   *  Constant: '<S427>/Constant'
   */
  if (rtb_RelationalOperator2_j) {
    rtb_MinMax_a = rtb_Divide4_d;
  } else {
    rtb_MinMax_a = 0.0;
  }

  /* End of Switch: '<S427>/Ign retard type 6' */

  /* Delay: '<S524>/Delay' incorporates:
   *  Constant: '<S427>/Constant2'
   *  Delay: '<S425>/Delay'
   */
  Gen2_ref_DWork->icLoad_dk = ((((Gen2_ref_PrevZCSigState->Delay_Reset_ZCE_h ==
    1) != (int32_T)rtb_bResetHlci) &&
    (Gen2_ref_PrevZCSigState->Delay_Reset_ZCE_h != 3)) || rtb_bResetHlci ||
    Gen2_ref_DWork->icLoad_dk);
  Gen2_ref_PrevZCSigState->Delay_Reset_ZCE_h = rtb_bResetHlci;
  if (Gen2_ref_DWork->icLoad_dk) {
    Gen2_ref_DWork->Delay_DSTATE_p = 0.0;
  }

  /* Switch: '<S524>/etaVolConst' incorporates:
   *  Constant: '<S427>/Constant2'
   */
  if (rtb_bResetHlci) {
    rtb_bResetHlci_0 = 0.0;
  } else {
    rtb_bResetHlci_0 = rtb_MinMax_a;
  }

  /* End of Switch: '<S524>/etaVolConst' */

  /* Sum: '<S524>/Difference Inputs1' incorporates:
   *  Delay: '<S524>/Delay'
   */
  rtb_Switch5_iq = rtb_bResetHlci_0 - Gen2_ref_DWork->Delay_DSTATE_p;

  /* Switch: '<S578>/Switch2' incorporates:
   *  RelationalOperator: '<S578>/LowerRelop1'
   */
  if (!(rtb_Switch5_iq > rtb_Sum1_dh)) {
    /* Product: '<S524>/delta fall limit' incorporates:
     *  Gain: '<S427>/Gain7'
     *  SampleTimeMath: '<S524>/sample time'
     *
     * About '<S524>/sample time':
     *  y = K where K = ( w * Ts )
     */
    rtb_Sum1_dh = -Gen2_ref_B->BusInput3.LR.rRateITadvance * 0.01;

    /* Switch: '<S578>/Switch' incorporates:
     *  RelationalOperator: '<S578>/UpperRelop'
     */
    if (!(rtb_Switch5_iq < rtb_Sum1_dh)) {
      rtb_Sum1_dh = rtb_Switch5_iq;
    }

    /* End of Switch: '<S578>/Switch' */
  }

  /* End of Switch: '<S578>/Switch2' */

  /* Sum: '<S524>/Difference Inputs2' incorporates:
   *  Delay: '<S524>/Delay'
   */
  rtb_Switch5_iq = rtb_Sum1_dh + Gen2_ref_DWork->Delay_DSTATE_p;

  /* MinMax: '<S427>/MinMax' */
  if ((rtb_Switch5_iq >= rtb_MinMax_a) || rtIsNaN(rtb_MinMax_a)) {
    rtb_MinMax_a = rtb_Switch5_iq;
  }

  /* End of MinMax: '<S427>/MinMax' */

  /* Gain: '<S9>/Gain5' */
  rtb_Sum1_dh = rtb_kW2W1_h;

  /* S-Function (sfix_look1_dyn): '<S9>/Lookup Table Dynamic1' */
  /* Dynamic Look-Up Table Block: '<S9>/Lookup Table Dynamic1'
   * Input0  Data Type:  Floating Point real_T
   * Input1  Data Type:  Floating Point real_T
   * Input2  Data Type:  Floating Point real_T
   * Output0 Data Type:  Floating Point real_T
   * Lookup Method: Linear_Endpoint
   *
   */
  LookUp_real_T_real_T( &(rtb_Switch_n),
                       &Gen2_ref_B->BusInput3.ITC.rITCoffsetP2s_y[0],
                       rtb_Sum1_dh, &Gen2_ref_B->BusInput3.ITC.rITCoffsetP2s_x[0],
                       4U, inst);

  /* Product: '<S811>/delta rise limit' */
  rtb_Sum1_dh = x;

  /* Delay: '<S811>/Delay' incorporates:
   *  Constant: '<S9>/Constant1'
   *  Delay: '<S425>/Delay'
   */
  Gen2_ref_DWork->icLoad_iv = ((((Gen2_ref_PrevZCSigState->Delay_Reset_ZCE_bi ==
    1) != (int32_T)rtb_bResetHlci) &&
    (Gen2_ref_PrevZCSigState->Delay_Reset_ZCE_bi != 3)) || rtb_bResetHlci ||
    Gen2_ref_DWork->icLoad_iv);
  Gen2_ref_PrevZCSigState->Delay_Reset_ZCE_bi = rtb_bResetHlci;
  if (Gen2_ref_DWork->icLoad_iv) {
    Gen2_ref_DWork->Delay_DSTATE_i4 = 0.0;
  }

  /* Switch: '<S811>/etaVolConst' incorporates:
   *  Constant: '<S9>/Constant1'
   */
  if (rtb_bResetHlci) {
    rtb_bResetHlci_0 = 0.0;
  } else {
    rtb_bResetHlci_0 = rtb_Switch_n;
  }

  /* End of Switch: '<S811>/etaVolConst' */

  /* Sum: '<S811>/Difference Inputs1' incorporates:
   *  Delay: '<S811>/Delay'
   */
  x = rtb_bResetHlci_0 - Gen2_ref_DWork->Delay_DSTATE_i4;

  /* Switch: '<S812>/Switch2' incorporates:
   *  RelationalOperator: '<S812>/LowerRelop1'
   */
  if (!(x > rtb_Sum1_dh)) {
    /* Product: '<S811>/delta fall limit' incorporates:
     *  Gain: '<S9>/Gain8'
     *  SampleTimeMath: '<S811>/sample time'
     *
     * About '<S811>/sample time':
     *  y = K where K = ( w * Ts )
     */
    rtb_Sum4_ny = -rtb_Sum4_ny * 0.01;

    /* Switch: '<S812>/Switch' incorporates:
     *  RelationalOperator: '<S812>/UpperRelop'
     */
    if (x < rtb_Sum4_ny) {
      rtb_Sum1_dh = rtb_Sum4_ny;
    } else {
      rtb_Sum1_dh = x;
    }

    /* End of Switch: '<S812>/Switch' */
  }

  /* End of Switch: '<S812>/Switch2' */

  /* Sum: '<S811>/Difference Inputs2' incorporates:
   *  Delay: '<S811>/Delay'
   */
  rtb_Sum4_ny = rtb_Sum1_dh + Gen2_ref_DWork->Delay_DSTATE_i4;

  /* MinMax: '<S9>/MinMax2' */
  if ((!(rtb_Switch_n >= rtb_Sum4_ny)) && (!rtIsNaN(rtb_Sum4_ny))) {
    rtb_Switch_n = rtb_Sum4_ny;
  }

  /* End of MinMax: '<S9>/MinMax2' */

  /* Sum: '<S9>/Sum1' incorporates:
   *  Gain: '<S9>/Gain'
   *  Gain: '<S9>/Gain3'
   *  Sum: '<S8>/Sum3'
   */
  rtb_Sum1_dh = -(rtb_Sum_c + rtb_MinMax_a) + -rtb_Switch_n;

  /* Switch: '<S9>/deltaIT' incorporates:
   *  Constant: '<S807>/Constant'
   *  Constant: '<S9>/Constant'
   *  RelationalOperator: '<S807>/Compare'
   */
  if (Gen2_ref_B->BusInput.iOpMode < 60) {
    rtb_Switch_n = 0.0;
  } else {
    rtb_Switch_n = rtb_Sum1_dh;
  }

  /* End of Switch: '<S9>/deltaIT' */

  /* Switch: '<S810>/Switch2' incorporates:
   *  RelationalOperator: '<S810>/LowerRelop1'
   */
  if (!(rtb_Switch_n > rtb_Divide2_f)) {
    /* Gain: '<S9>/Gain4' incorporates:
     *  Abs: '<S9>/Abs'
     */
    rtb_Divide2_f = -fabs(Gen2_ref_B->BusInput3.ITC.rITCdeltaMIN);

    /* Switch: '<S810>/Switch' incorporates:
     *  RelationalOperator: '<S810>/UpperRelop'
     */
    if (!(rtb_Switch_n < rtb_Divide2_f)) {
      rtb_Divide2_f = rtb_Switch_n;
    }

    /* End of Switch: '<S810>/Switch' */
  }

  /* End of Switch: '<S810>/Switch2' */

  /* BusCreator: '<S16>/Bus Creator' incorporates:
   *  DataTypeConversion: '<S16>/Data Type Conversion10'
   *  Outport: '<Root>/out'
   */
  Gen2_ref_Y->out.rdeltaIT = (real32_T)rtb_Divide2_f;

  /* Gain: '<S16>/W2kW' */
  rtb_Divide2_f = rtb_PactOut_tmp;

  /* BusCreator: '<S16>/Bus Creator' incorporates:
   *  DataTypeConversion: '<S16>/Data Type Conversion4'
   *  Outport: '<Root>/out'
   */
  Gen2_ref_Y->out.rP_des = (real32_T)rtb_Divide2_f;

  /* Switch: '<S14>/Switch1' */
  for (i = 0; i < 10; i++) {
    if (Gen2_ref_B->BusInput3.LamLim.bNOx250mg) {
      Gen2_ref_Y->out.rLamMap[i] = Gen2_ref_B->
        BusInput3.LamLim.rLamMapBase250mg[i];
    } else {
      Gen2_ref_Y->out.rLamMap[i] = Gen2_ref_B->BusInput3.LamLim.rLamMapBase[i];
    }
  }

  /* End of Switch: '<S14>/Switch1' */

  /* DataTypeConversion: '<S16>/Data Type Conversion21' */
  for (i = 0; i < 13; i++) {
    Gen2_ref_Y->out.rState_Dist1Map[i] = (real32_T)rtb_y_map_new[i];
  }

  /* End of DataTypeConversion: '<S16>/Data Type Conversion21' */

  /* Switch: '<S12>/Switch7' */
  if (Gen2_ref_B->BusInput3.SpeedCtrl.bUseFilteredFeedback) {
    rtb_Divide2_f = Gen2_ref_B->p2s_filt.Switch;
  } else {
    rtb_Divide2_f = rtb_p2s;
  }

  /* End of Switch: '<S12>/Switch7' */

  /* Gain: '<S815>/Gain6' incorporates:
   *  Gain: '<S12>/Gain3'
   */
  rtb_kW2W1_h = 1.0E-5 * rtb_Divide2_f;

  /* Switch: '<S814>/Switch3' */
  if (Gen2_ref_B->BusInput3.SpeedCtrl.bMeasPowKeEst) {
    rtb_Switch_n = rtb_Gain2_ao;
  } else {
    rtb_Switch_n = rtb_kW2W;
  }

  /* End of Switch: '<S814>/Switch3' */

  /* Gain: '<S814>/Gain10' */
  x = rtb_Switch2_ejy_tmp;

  /* Sum: '<S814>/Sum3' */
  rtb_kW2W = rtb_Switch_n + x;

  /* Gain: '<S814>/Gain11' */
  rtb_Switch_n = 0.10471975511965977 * rtb_DataTypeConversion15;

  /* Abs: '<S820>/Abs' */
  x = fabs(rtb_Switch_n);

  /* Switch: '<S820>/Switch' incorporates:
   *  Constant: '<S820>/Constant2'
   *  RelationalOperator: '<S820>/Relational Operator'
   */
  if (2.2204460492503131E-16 >= x) {
    rtb_bResetHlci_0 = 2.2204460492503131E-16;
  } else {
    rtb_bResetHlci_0 = rtb_Switch_n;
  }

  /* End of Switch: '<S820>/Switch' */

  /* Gain: '<S12>/Gain3' */
  x = rtb_kW2W1_h;

  /* Product: '<S814>/Divide5' */
  rtb_Divide2_f = rtb_Product1_fu * rtb_Sum1_idx_2;

  /* Sum: '<S814>/Sum4' incorporates:
   *  Constant: '<S814>/it_offset_ref2'
   */
  rtb_Divide2_f++;

  /* Abs: '<S821>/Abs' */
  rtb_Switch_n = fabs(rtb_Divide2_f);

  /* Switch: '<S821>/Switch' incorporates:
   *  Constant: '<S821>/Constant2'
   *  RelationalOperator: '<S821>/Relational Operator'
   */
  if (2.2204460492503131E-16 >= rtb_Switch_n) {
    rtb_Divide2_f = 2.2204460492503131E-16;
  }

  /* End of Switch: '<S821>/Switch' */

  /* Product: '<S814>/Divide4' */
  rtb_Divide2_f = x / rtb_Divide2_f;

  /* Abs: '<S822>/Abs' */
  rtb_Switch_n = fabs(rtb_Divide2_f);

  /* Switch: '<S822>/Switch' incorporates:
   *  Constant: '<S822>/Constant2'
   *  RelationalOperator: '<S822>/Relational Operator'
   */
  if (2.2204460492503131E-16 >= rtb_Switch_n) {
    rtb_Divide2_f = 2.2204460492503131E-16;
  }

  /* End of Switch: '<S822>/Switch' */

  /* Outputs for Atomic SubSystem: '<S814>/Filter1' */
  /* Product: '<S814>/Divide11' incorporates:
   *  Product: '<S814>/Divide3'
   */
  Gen2_ref_N_TC_HP_filt(rtb_kW2W / rtb_bResetHlci_0 / rtb_Divide2_f,
                        Gen2_ref_B->BusInput3.SpeedCtrl.rTiFKeEst,
                        rtb_LogicalOperator_cn, &Gen2_ref_B->Filter1_n,
                        &Gen2_ref_DWork->Filter1_n, inst);

  /* End of Outputs for SubSystem: '<S814>/Filter1' */

  /* Abs: '<S817>/Abs' */
  rtb_Divide2_f = delta_y;

  /* Switch: '<S817>/Switch' incorporates:
   *  Constant: '<S817>/Constant2'
   *  RelationalOperator: '<S817>/Relational Operator'
   */
  if (2.2204460492503131E-16 >= rtb_Divide2_f) {
    delta_y = 2.2204460492503131E-16;
  } else {
    delta_y = Gen2_ref_B->T2s_filt.Switch;
  }

  /* End of Switch: '<S817>/Switch' */

  /* Product: '<S5>/Divide4' incorporates:
   *  Product: '<S268>/Divide3'
   */
  rtb_Switch_n = rtb_Switch_ks * Gen2_ref_B->BusInput.IN_EC_rGT_RatioMix_TC2;

  /* Sum: '<S5>/Add3' incorporates:
   *  Constant: '<S11>/Constant'
   *  Sum: '<S11>/Sum'
   */
  x = 1.0 - Gen2_ref_B->BusInput.IN_EC_rGT_RatioMix_TC2;

  /* Sum: '<S5>/Add4' incorporates:
   *  Product: '<S267>/Divide3'
   *  Product: '<S5>/Divide5'
   */
  rtb_kW2W = rtb_Divide3_n_tmp * x + rtb_Switch_n;

  /* Abs: '<S816>/Abs' */
  rtb_Switch_n = fabs(rtb_kW2W);

  /* Saturate: '<S813>/Saturation' */
  if (Gen2_ref_B->BusInput3.eng.rNum_Cyl_Eng <= 1.0) {
    rtb_Divide2_f = 1.0;
  } else {
    rtb_Divide2_f = Gen2_ref_B->BusInput3.eng.rNum_Cyl_Eng;
  }

  /* End of Saturate: '<S813>/Saturation' */

  /* Product: '<S813>/Divide1' */
  u0 = 1.0 / rtb_Divide2_f * r;

  /* Switch: '<S816>/Switch' incorporates:
   *  Constant: '<S816>/Constant2'
   *  RelationalOperator: '<S816>/Relational Operator'
   */
  if (2.2204460492503131E-16 >= rtb_Switch_n) {
    rtb_bResetHlci_0 = 2.2204460492503131E-16;
  } else {
    rtb_bResetHlci_0 = rtb_kW2W;
  }

  /* End of Switch: '<S816>/Switch' */

  /* Saturate: '<S813>/Saturation1' */
  if (u0 > 1.0) {
    u0 = 1.0;
  } else if (u0 < 0.0) {
    u0 = 0.0;
  }

  /* End of Saturate: '<S813>/Saturation1' */

  /* Product: '<S813>/Product' incorporates:
   *  Constant: '<S813>/it_offset_ref2'
   *  Gain: '<S813>/Gain1'
   *  Gain: '<S813>/Gain2'
   *  Product: '<S813>/Divide3'
   *  Sum: '<S813>/Sum3'
   */
  r = Gen2_ref_B->BusInput3.eng.rVol_Hub_Eng / delta_y * rtb_etaVolConst_lt *
    rtb_etaBreakConst * rtb_Sum1_idx_3 / rtb_bResetHlci_0 * 0.079577471545947673
    * 100000.0 * (1.0 - u0);

  /* Abs: '<S834>/Abs' */
  rtb_Divide2_f = fabs(r);

  /* Switch: '<S834>/Switch' incorporates:
   *  Constant: '<S834>/Constant2'
   *  RelationalOperator: '<S834>/Relational Operator'
   */
  if (2.2204460492503131E-16 >= rtb_Divide2_f) {
    rtb_bResetHlci_0 = 2.2204460492503131E-16;
  } else {
    rtb_bResetHlci_0 = r;
  }

  /* End of Switch: '<S834>/Switch' */

  /* Product: '<S830>/Product1' */
  rtb_Switch_n = Gen2_ref_B->Filter1_n.Switch / rtb_bResetHlci_0;

  /* Logic: '<S830>/Logical Operator2' */
  rtb_LogicalOperator2_l = (rtb_LogicalOperator_cn || rtb_LogicalOperator2_l);

  /* Delay: '<S830>/Resettable Delay' */
  Gen2_ref_DWork->icLoad_ix = ((rtb_LogicalOperator2_l &&
    (Gen2_ref_PrevZCSigState->ResettableDelay_Reset_ZCE_k != 1)) ||
    Gen2_ref_DWork->icLoad_ix);
  Gen2_ref_PrevZCSigState->ResettableDelay_Reset_ZCE_k = rtb_LogicalOperator2_l;
  for (i = 0; i < 13; i++) {
    if (Gen2_ref_DWork->icLoad_ix) {
      Gen2_ref_DWork->ResettableDelay_DSTATE_k[i] =
        Gen2_ref_B->BusInput3.SpeedCtrl.refPoint_iLQR_Keng_y[i];
    }

    rtb_Switch3_je[i] = Gen2_ref_DWork->ResettableDelay_DSTATE_k[i];
  }

  /* End of Delay: '<S830>/Resettable Delay' */

  /* S-Function (sfix_look1_dyn): '<S830>/gain scheduling Keng1' */
  /* Dynamic Look-Up Table Block: '<S830>/gain scheduling Keng1'
   * Input0  Data Type:  Floating Point real_T
   * Input1  Data Type:  Floating Point real_T
   * Input2  Data Type:  Floating Point real_T
   * Output0 Data Type:  Floating Point real_T
   * Lookup Method: Linear_Endpoint
   *
   */
  LookUp_real_T_real_T( &(rtb_gainschedulingKeng1_f), &rtb_Switch3_je[0],
                       rtb_kW2W1_h,
                       &Gen2_ref_B->BusInput3.SpeedCtrl.refPoint_iLQR_Keng_x[0],
                       12U, inst);

  /* Outputs for Atomic SubSystem: '<S831>/TP' */
  /* UnitDelay: '<S831>/Unit Delay2' incorporates:
   *  SignalConversion generated from: '<S831>/Bus Selector1'
   */
  Gen2_ref_TP(Gen2_ref_DWork->UnitDelay2_DSTATE_i,
              Gen2_ref_B->BusInput3.SpeedCtrl.rTp_KeEst_reset, &Gen2_ref_B->TP_g,
              &Gen2_ref_DWork->TP_g, inst);

  /* End of Outputs for SubSystem: '<S831>/TP' */

  /* Outputs for Atomic SubSystem: '<S831>/TON1' */
  Gen2_ref_TON_1(Gen2_ref_DWork->UnitDelay2_DSTATE_i,
                 Gen2_ref_B->BusInput3.SpeedCtrl.tOutOfNWindow,
                 &Gen2_ref_B->TON1_m, &Gen2_ref_DWork->TON1_m, inst);

  /* End of Outputs for SubSystem: '<S831>/TON1' */

  /* Outputs for Atomic SubSystem: '<S831>/TP1' */
  Gen2_ref_TP(Gen2_ref_DWork->UnitDelay2_DSTATE_i,
              Gen2_ref_B->BusInput3.SpeedCtrl.rT_KeEstIncreaseTiF,
              &Gen2_ref_B->TP1_l, &Gen2_ref_DWork->TP1_l, inst);

  /* End of Outputs for SubSystem: '<S831>/TP1' */

  /* UnitDelay: '<S831>/Unit Delay1' */
  rtb_Divide2_f = Gen2_ref_DWork->UnitDelay1_DSTATE_n;

  /* DataTypeConversion: '<S831>/Data Type Conversion' */
  rtb_bResetHlci_0 = floor(rtb_Divide2_f);
  if (rtIsNaN(rtb_bResetHlci_0) || rtIsInf(rtb_bResetHlci_0)) {
    rtb_bResetHlci_0 = 0.0;
  } else {
    rtb_bResetHlci_0 = fmod(rtb_bResetHlci_0, 65536.0);
  }

  /* Outputs for Atomic SubSystem: '<S831>/TOF' */
  /* RelationalOperator: '<S831>/Relational Operator' incorporates:
   *  DataTypeConversion: '<S831>/Data Type Conversion'
   */
  Gen2_ref_TOF(((rtb_bResetHlci_0 < 0.0 ? (int32_T)(int16_T)-(int16_T)(uint16_T)
                 -rtb_bResetHlci_0 : (int32_T)(int16_T)(uint16_T)
                 rtb_bResetHlci_0) > 0),
               Gen2_ref_B->BusInput3.SpeedCtrl.rTof_KeEstPause_SkipF,
               &Gen2_ref_B->TOF_n, &Gen2_ref_DWork->TOF_n, inst);

  /* End of Outputs for SubSystem: '<S831>/TOF' */

  /* Switch: '<S831>/Switch3' incorporates:
   *  Constant: '<S831>/Constant2'
   *  Switch: '<S831>/Switch1'
   */
  if (Gen2_ref_B->BusInput3.SpeedCtrl.bKeEstIncreaseTiFOFF) {
    rtb_Switch3_le = false;
  } else if (Gen2_ref_B->BusInput3.SpeedCtrl.bKeEstPause_SkipF) {
    /* Switch: '<S831>/Switch1' incorporates:
     *  Logic: '<S831>/Logical Operator3'
     */
    rtb_Switch3_le = (Gen2_ref_B->TP1_l.LogicalOperator1 ||
                      Gen2_ref_B->TOF_n.LogicalOperator1);
  } else {
    /* Switch: '<S831>/Switch1' */
    rtb_Switch3_le = Gen2_ref_B->TP1_l.LogicalOperator1;
  }

  /* End of Switch: '<S831>/Switch3' */

  /* Switch: '<S831>/Switch2' incorporates:
   *  Constant: '<S831>/Constant1'
   *  Logic: '<S831>/Logical Operator4'
   *  Logic: '<S831>/Logical Operator5'
   *  Switch: '<S831>/Switch'
   *  UnitDelay: '<S831>/Unit Delay2'
   */
  if (Gen2_ref_B->BusInput3.SpeedCtrl.bKeEstResetOFF) {
    rtb_LogicalOperator2_ov = false;
  } else if (Gen2_ref_B->BusInput3.SpeedCtrl.bKeEstreset_TP) {
    /* Switch: '<S831>/Switch' */
    rtb_LogicalOperator2_ov = Gen2_ref_B->TP_g.LogicalOperator1;
  } else {
    rtb_LogicalOperator2_ov = (Gen2_ref_DWork->UnitDelay2_DSTATE_i &&
      (!Gen2_ref_B->TON1_m.LogicalOperator3));
  }

  /* End of Switch: '<S831>/Switch2' */

  /* Outputs for Atomic SubSystem: '<S830>/Ke Map Update' */
  Gen2_ref_KeMapUpdate(rtb_Switch_n, rtb_LogicalOperator_cn,
                       rtb_gainschedulingKeng1_f, rtb_Switch3_le,
                       rtb_LogicalOperator2_ov, &Gen2_ref_B->BusInput3,
                       &Gen2_ref_B->KeMapUpdate_h,
                       &Gen2_ref_DWork->KeMapUpdate_h, inst);

  /* End of Outputs for SubSystem: '<S830>/Ke Map Update' */

  /* Switch: '<S830>/Switch1' incorporates:
   *  Logic: '<S830>/Logical Operator4'
   */
  if (Gen2_ref_B->BusInput3.SpeedCtrl.bActKeEst2Dof) {
    rtb_Switch_n = Gen2_ref_B->KeMapUpdate_h.Sum1;
  }

  /* End of Switch: '<S830>/Switch1' */

  /* MATLAB Function: '<S830>/MATLAB Function1' incorporates:
   *  Delay: '<S830>/Delay'
   *  Logic: '<S830>/Logical Operator1'
   */
  Gen2_ref_MATLABFunction1_m
    (Gen2_ref_B->BusInput3.SpeedCtrl.refPoint_iLQR_Keng_x,
     Gen2_ref_B->BusInput3.SpeedCtrl.refPoint_iLQR_Keng_y,
     Gen2_ref_B->BusInput3.SpeedCtrl.rKeAdaptEps, rtb_kW2W1_h, rtb_Switch_n,
     Gen2_ref_DWork->Delay_DSTATE_n2, !rtb_Switch3_le,
     &Gen2_ref_B->sf_MATLABFunction1_l, &Gen2_ref_DWork->sf_MATLABFunction1_l, inst);

  /* Logic: '<Root>/Logical Operator3' */
  rtb_bTV_sat = (Gen2_ref_B->BusInput3.KeEstNetP.bActKeEstNetP &&
                 rtb_LogicalOperator);

  /* MATLAB Function: '<S666>/MATLAB Function1' incorporates:
   *  Delay: '<S666>/Delay'
   *  Logic: '<S666>/Logical Operator1'
   */
  Gen2_ref_MATLABFunction1_m
    (Gen2_ref_B->BusInput3.SpeedCtrl.refPoint_iLQR_Keng_x,
     Gen2_ref_B->BusInput3.SpeedCtrl.refPoint_iLQR_Keng_y,
     Gen2_ref_B->BusInput3.SpeedCtrl.rKeAdaptEps, rtb_Gain6_b, rtb_Switch1_ep,
     Gen2_ref_DWork->Delay_DSTATE_cnq, !rtb_Switch3_of,
     &Gen2_ref_B->sf_MATLABFunction1_m, &Gen2_ref_DWork->sf_MATLABFunction1_m, inst);

  /* Sum: '<S635>/Sum' incorporates:
   *  Delay: '<S637>/Resettable Delay'
   */
  rtb_kW2W1_h = Gen2_ref_DWork->ResettableDelay_DSTATE_i - rtb_Switch1_k;

  /* Abs: '<S635>/Abs1' */
  rtb_Divide2_f = fabs(Gen2_ref_B->BusInput3.LamLim.rThrshLamSatOn);

  /* Abs: '<S635>/Abs' */
  rtb_Switch_n = fabs(Gen2_ref_B->BusInput3.LamLim.rThrshLamSatOff);

  /* MinMax: '<S635>/MinMax' */
  if ((rtb_Divide2_f >= rtb_Switch_n) || rtIsNaN(rtb_Switch_n)) {
    rtb_Gain6_b = rtb_Divide2_f;
  } else {
    rtb_Gain6_b = rtb_Switch_n;
  }

  /* End of MinMax: '<S635>/MinMax' */

  /* Switch: '<S635>/Switch2' incorporates:
   *  Constant: '<S635>/Constant4'
   *  RelationalOperator: '<S635>/Relational Operator'
   *  RelationalOperator: '<S635>/Relational Operator1'
   *  Switch: '<S635>/Switch3'
   *  UnitDelay: '<S635>/Unit Delay1'
   */
  if (rtb_kW2W1_h < rtb_Divide2_f) {
    rtb_kW2W1_h = 1.0;
  } else if (rtb_kW2W1_h > rtb_Gain6_b) {
    /* Switch: '<S635>/Switch3' incorporates:
     *  Constant: '<S635>/Constant5'
     */
    rtb_kW2W1_h = 0.0;
  } else {
    rtb_kW2W1_h = Gen2_ref_DWork->UnitDelay1_DSTATE_eq;
  }

  /* End of Switch: '<S635>/Switch2' */

  /* Sum: '<S635>/Sum1' incorporates:
   *  Delay: '<S637>/Resettable Delay'
   */
  rtb_Switch1_ep = rtb_Switch2_n5 - Gen2_ref_DWork->ResettableDelay_DSTATE_i;

  /* Switch: '<S635>/Switch4' incorporates:
   *  Constant: '<S635>/Constant6'
   *  RelationalOperator: '<S635>/Relational Operator2'
   *  RelationalOperator: '<S635>/Relational Operator3'
   *  Switch: '<S635>/Switch5'
   *  UnitDelay: '<S635>/Unit Delay2'
   */
  if (rtb_Switch1_ep < rtb_Divide2_f) {
    rtb_Gain6_b = 1.0;
  } else if (rtb_Switch1_ep > rtb_Gain6_b) {
    /* Switch: '<S635>/Switch5' incorporates:
     *  Constant: '<S635>/Constant7'
     */
    rtb_Gain6_b = 0.0;
  } else {
    rtb_Gain6_b = Gen2_ref_DWork->UnitDelay2_DSTATE_di;
  }

  /* End of Switch: '<S635>/Switch4' */

  /* Logic: '<S635>/Logical Operator2' */
  rtb_LogicalOperator2_ov = ((rtb_kW2W1_h != 0.0) || (rtb_Gain6_b != 0.0));

  /* Switch: '<S714>/Switch7' incorporates:
   *  Constant: '<S714>/Constant1'
   *  Logic: '<S714>/Logical Operator5'
   */
  if (!rtb_LogicalOperator2_ov) {
    rtb_Divide2_f = Gen2_ref_B->BusInput3.SpeedCtrl.rKeAdaptEps;
  } else {
    rtb_Divide2_f = 0.0;
  }

  /* End of Switch: '<S714>/Switch7' */

  /* Outputs for Atomic SubSystem: '<S714>/TON' */
  Gen2_ref_TON_1(Gen2_ref_B->TON2.LogicalOperator3,
                 Gen2_ref_B->BusInput3.SpeedCtrl.rKeAdaptTon, &Gen2_ref_B->TON_o,
                 &Gen2_ref_DWork->TON_o, inst);

  /* End of Outputs for SubSystem: '<S714>/TON' */

  /* Logic: '<S714>/Logical Operator1' */
  rtb_Switch2_au = (rtb_RelationalOperator_ok &&
                    Gen2_ref_B->TON_o.LogicalOperator3);

  /* MATLAB Function: '<S714>/MATLAB Function1' incorporates:
   *  Delay: '<S714>/Delay'
   */
  if ((!Gen2_ref_DWork->y_map_not_empty_d) || Gen2_ref_DWork->Delay_DSTATE_a) {
    Gen2_ref_DWork->y_map_not_empty_d = true;
    for (i = 0; i < 13; i++) {
      Gen2_ref_DWork->y_map_f[i] =
        Gen2_ref_B->BusInput3.SpeedCtrl.refPoint_iLQR_Keng_y[i];
      Gen2_ref_DWork->x_map_n[i] =
        Gen2_ref_B->BusInput3.SpeedCtrl.refPoint_iLQR_Keng_x[i];
    }
  }

  if (Gen2_ref_maximum_f(Gen2_ref_DWork->y_map_f, inst) < 0.1) {
    for (i = 0; i < 13; i++) {
      Gen2_ref_DWork->y_map_f[i] =
        Gen2_ref_B->BusInput3.SpeedCtrl.refPoint_iLQR_Keng_y[i];
    }
  }

  if (!rtIsNaN(Gen2_ref_DWork->x_map_n[0])) {
    k = 1;
  } else {
    k = 0;
    i = 2;
    exitg1 = false;
    while ((!exitg1) && (i < 14)) {
      if (!rtIsNaN(Gen2_ref_DWork->x_map_n[i - 1])) {
        k = i;
        exitg1 = true;
      } else {
        i++;
      }
    }
  }

  if (k == 0) {
    rtb_Switch1_ep = Gen2_ref_DWork->x_map_n[0];
  } else {
    rtb_Switch1_ep = Gen2_ref_DWork->x_map_n[k - 1];
    while (k + 1 <= 13) {
      if (rtb_Switch1_ep > Gen2_ref_DWork->x_map_n[k]) {
        rtb_Switch1_ep = Gen2_ref_DWork->x_map_n[k];
      }

      k++;
    }
  }

  if ((rtb_Switch1_ep >= rtb_Gain6_jx) || rtIsNaN(rtb_Gain6_jx)) {
    rtb_Gain6_jx = rtb_Switch1_ep;
  }

  x = Gen2_ref_maximum_f(Gen2_ref_DWork->x_map_n, inst);
  if ((!(x <= rtb_Gain6_jx)) && (!rtIsNaN(rtb_Gain6_jx))) {
    x = rtb_Gain6_jx;
  }

  k = 0;
  if (!(x < Gen2_ref_DWork->x_map_n[0])) {
    for (i = 0; i < 13; i++) {
      if (x > Gen2_ref_DWork->x_map_n[i]) {
        k = i;
      }
    }
  }

  if (k + 1 < 13) {
    if (rtb_Switch2_au && (!Gen2_ref_DWork->Delay_DSTATE_a)) {
      rtb_Switch_n = Gen2_ref_DWork->y_map_f[k + 1];
      delta_y_tmp_tmp = x - Gen2_ref_DWork->x_map_n[k];
      u0 = Gen2_ref_DWork->x_map_n[k + 1];
      delta_y = delta_y_tmp_tmp / (u0 - Gen2_ref_DWork->x_map_n[k]) *
        (rtb_Switch_n - Gen2_ref_DWork->y_map_f[k]) + Gen2_ref_DWork->y_map_f[k];
      delta_y = ((1.0 - rtb_Divide2_f) * delta_y + rtb_Divide2_f * rtb_Sum_ig) -
        delta_y;
      x = u0 - x;
      rtb_Divide2_f = delta_y_tmp_tmp + x;
      rtb_PactOut_tmp = rtb_Divide2_f * x;
      rtb_bResetHlci_0 = (delta_y_tmp_tmp * delta_y_tmp_tmp + rtb_PactOut_tmp) -
        delta_y_tmp_tmp * x;
      Gen2_ref_DWork->y_map_f[k] += rtb_PactOut_tmp * delta_y / rtb_bResetHlci_0;
      Gen2_ref_DWork->y_map_f[k + 1] = rtb_Divide2_f * delta_y_tmp_tmp * delta_y
        / rtb_bResetHlci_0 + rtb_Switch_n;
    }
  } else if (rtb_Switch2_au && (!Gen2_ref_DWork->Delay_DSTATE_a)) {
    Gen2_ref_DWork->y_map_f[12] = (1.0 - rtb_Divide2_f) *
      Gen2_ref_DWork->y_map_f[12] + rtb_Divide2_f * rtb_Sum_ig;
  }

  for (i = 0; i < 13; i++) {
    rtb_y_map_new_n[i] = Gen2_ref_DWork->y_map_f[i];
  }

  /* Switch: '<S431>/Switch3' incorporates:
   *  MATLAB Function: '<S714>/MATLAB Function1'
   */
  for (i = 0; i < 13; i++) {
    if (Gen2_ref_B->BusInput3.SpeedCtrl.bActKeEstMapUpdate) {
      rtb_Switch3_je[i] = Gen2_ref_B->sf_MATLABFunction1_m.y_map_new[i];
    } else {
      rtb_Switch3_je[i] = Gen2_ref_DWork->y_map_f[i];
    }
  }

  /* End of Switch: '<S431>/Switch3' */

  /* Switch: '<S715>/Switch7' incorporates:
   *  Constant: '<S715>/Constant1'
   *  Logic: '<S715>/Logical Operator5'
   */
  if (!rtb_LogicalOperator2_ov) {
    rtb_Divide2_f = Gen2_ref_B->BusInput3.SpeedCtrl.rKeAdaptEps;
  } else {
    rtb_Divide2_f = 0.0;
  }

  /* End of Switch: '<S715>/Switch7' */

  /* Outputs for Atomic SubSystem: '<S715>/TON' */
  Gen2_ref_TON_1(Gen2_ref_B->TON2.LogicalOperator3,
                 Gen2_ref_B->BusInput3.SpeedCtrl.rKeAdaptTon, &Gen2_ref_B->TON_m,
                 &Gen2_ref_DWork->TON_m, inst);

  /* End of Outputs for SubSystem: '<S715>/TON' */

  /* Logic: '<S715>/Logical Operator1' incorporates:
   *  Logic: '<S636>/Logical Operator'
   */
  rtb_Switch3_le = ((!rtb_RelationalOperator_ok) &&
                    Gen2_ref_B->TON_m.LogicalOperator3);

  /* MATLAB Function: '<S715>/MATLAB Function1' incorporates:
   *  Delay: '<S715>/Delay'
   */
  if ((!Gen2_ref_DWork->y_map_not_empty_f) || Gen2_ref_DWork->Delay_DSTATE_ng) {
    Gen2_ref_DWork->y_map_not_empty_f = true;
    for (i = 0; i < 7; i++) {
      Gen2_ref_DWork->y_map_i[i] =
        Gen2_ref_B->BusInput3.SpeedCtrl.refPoint_iLQR_KengPOW_y[i];
      Gen2_ref_DWork->x_map_c[i] =
        Gen2_ref_B->BusInput3.SpeedCtrl.refPoint_iLQR_KengPOW_x[i];
    }
  }

  if (Gen2_ref_maximum_f5(Gen2_ref_DWork->y_map_i, inst) < 0.1) {
    for (i = 0; i < 7; i++) {
      Gen2_ref_DWork->y_map_i[i] =
        Gen2_ref_B->BusInput3.SpeedCtrl.refPoint_iLQR_KengPOW_y[i];
    }
  }

  if (!rtIsNaN(Gen2_ref_DWork->x_map_c[0])) {
    k = 1;
  } else {
    k = 0;
    i = 2;
    exitg1 = false;
    while ((!exitg1) && (i < 8)) {
      if (!rtIsNaN(Gen2_ref_DWork->x_map_c[i - 1])) {
        k = i;
        exitg1 = true;
      } else {
        i++;
      }
    }
  }

  if (k == 0) {
    rtb_Switch1_ep = Gen2_ref_DWork->x_map_c[0];
  } else {
    rtb_Switch1_ep = Gen2_ref_DWork->x_map_c[k - 1];
    while (k + 1 <= 7) {
      if (rtb_Switch1_ep > Gen2_ref_DWork->x_map_c[k]) {
        rtb_Switch1_ep = Gen2_ref_DWork->x_map_c[k];
      }

      k++;
    }
  }

  if ((rtb_Switch1_ep >= rtb_Gain7) || rtIsNaN(rtb_Gain7)) {
    rtb_Gain7 = rtb_Switch1_ep;
  }

  x = Gen2_ref_maximum_f5(Gen2_ref_DWork->x_map_c, inst);
  if ((!(x <= rtb_Gain7)) && (!rtIsNaN(rtb_Gain7))) {
    x = rtb_Gain7;
  }

  k = 0;
  if (!(x < Gen2_ref_DWork->x_map_c[0])) {
    for (i = 0; i < 7; i++) {
      if (x > Gen2_ref_DWork->x_map_c[i]) {
        k = i;
      }
    }
  }

  if (k + 1 < 7) {
    if (rtb_Switch3_le && (!Gen2_ref_DWork->Delay_DSTATE_ng)) {
      rtb_Switch_n = Gen2_ref_DWork->y_map_i[k + 1];
      delta_y_tmp_tmp = x - Gen2_ref_DWork->x_map_c[k];
      u0 = Gen2_ref_DWork->x_map_c[k + 1];
      delta_y = delta_y_tmp_tmp / (u0 - Gen2_ref_DWork->x_map_c[k]) *
        (rtb_Switch_n - Gen2_ref_DWork->y_map_i[k]) + Gen2_ref_DWork->y_map_i[k];
      delta_y = ((1.0 - rtb_Divide2_f) * delta_y + rtb_Divide2_f * rtb_Sum_gb) -
        delta_y;
      x = u0 - x;
      rtb_Divide2_f = delta_y_tmp_tmp + x;
      rtb_PactOut_tmp = rtb_Divide2_f * x;
      rtb_Gain7 = (delta_y_tmp_tmp * delta_y_tmp_tmp + rtb_PactOut_tmp) -
        delta_y_tmp_tmp * x;
      Gen2_ref_DWork->y_map_i[k] += rtb_PactOut_tmp * delta_y / rtb_Gain7;
      Gen2_ref_DWork->y_map_i[k + 1] = rtb_Divide2_f * delta_y_tmp_tmp * delta_y
        / rtb_Gain7 + rtb_Switch_n;
    }
  } else if (rtb_Switch3_le && (!Gen2_ref_DWork->Delay_DSTATE_ng)) {
    Gen2_ref_DWork->y_map_i[6] = (1.0 - rtb_Divide2_f) * Gen2_ref_DWork->
      y_map_i[6] + rtb_Divide2_f * rtb_Sum_gb;
  }

  for (i = 0; i < 7; i++) {
    rtb_y_map_new_a[i] = Gen2_ref_DWork->y_map_i[i];
  }

  /* Sum: '<S275>/Add2' incorporates:
   *  Sum: '<S291>/Add2'
   */
  rtb_PactOut_tmp = Gen2_ref_B->BusInput3.leanox.rP_Eng_Frict +
    Gen2_ref_B->BusInput3.eng.rP_Nom;
  rtb_Divide2_f = rtb_PactOut_tmp;

  /* Gain: '<S275>/Gain' */
  rtb_Gain7 = 1000.0 * rtb_Divide2_f;

  /* Abs: '<S281>/Abs' */
  rtb_Divide2_f = fabs(Gen2_ref_B->BusInput3.eng.rLHV);

  /* Abs: '<S282>/Abs' incorporates:
   *  Abs: '<S298>/Abs'
   */
  rtb_Switch_n = fabs(Gen2_ref_B->BusInput3.Eff.rEtaBrakeExt);

  /* Switch: '<S281>/Switch' incorporates:
   *  Constant: '<S281>/Constant2'
   *  RelationalOperator: '<S281>/Relational Operator'
   */
  if (2.2204460492503131E-16 >= rtb_Divide2_f) {
    rtb_bResetHlci_0 = 2.2204460492503131E-16;
  } else {
    rtb_bResetHlci_0 = Gen2_ref_B->BusInput3.eng.rLHV;
  }

  /* End of Switch: '<S281>/Switch' */

  /* Switch: '<S282>/Switch' incorporates:
   *  Constant: '<S282>/Constant2'
   *  RelationalOperator: '<S282>/Relational Operator'
   */
  if (2.2204460492503131E-16 >= rtb_Switch_n) {
    delta_y = 2.2204460492503131E-16;
  } else {
    delta_y = Gen2_ref_B->BusInput3.Eff.rEtaBrakeExt;
  }

  /* End of Switch: '<S282>/Switch' */

  /* Product: '<S275>/Divide4' */
  rtb_Divide2_f = rtb_Gain7 / rtb_bResetHlci_0 / delta_y;

  /* Gain: '<S275>/Gain3' */
  rtb_Gain7 = 0.1 * rtb_Divide2_f;

  /* BusCreator: '<S16>/Bus Creator' incorporates:
   *  Outport: '<Root>/out'
   *  RelationalOperator: '<S275>/Relational Operator'
   *  Sum: '<S275>/Add3'
   */
  Gen2_ref_Y->out.TJ_GasO[1] = (rtb_SumofElements > rtb_Divide2_f + rtb_Gain7);

  /* Sum: '<S291>/Add2' */
  rtb_Divide2_f = rtb_PactOut_tmp;

  /* Gain: '<S291>/Gain' */
  rtb_Sum_gb = 1000.0 * rtb_Divide2_f;

  /* Abs: '<S297>/Abs' */
  rtb_Divide2_f = fabs(Gen2_ref_B->BusInput3.eng.rLHV_M);

  /* Switch: '<S297>/Switch' incorporates:
   *  Constant: '<S297>/Constant2'
   *  RelationalOperator: '<S297>/Relational Operator'
   */
  if (2.2204460492503131E-16 >= rtb_Divide2_f) {
    rtb_bResetHlci_0 = 2.2204460492503131E-16;
  } else {
    rtb_bResetHlci_0 = Gen2_ref_B->BusInput3.eng.rLHV_M;
  }

  /* End of Switch: '<S297>/Switch' */

  /* Switch: '<S298>/Switch' incorporates:
   *  Constant: '<S298>/Constant2'
   *  RelationalOperator: '<S298>/Relational Operator'
   */
  if (2.2204460492503131E-16 >= rtb_Switch_n) {
    delta_y = 2.2204460492503131E-16;
  } else {
    delta_y = Gen2_ref_B->BusInput3.Eff.rEtaBrakeExt;
  }

  /* End of Switch: '<S298>/Switch' */

  /* Product: '<S291>/Divide4' */
  rtb_Divide2_f = rtb_Sum_gb / rtb_bResetHlci_0 / delta_y;

  /* Gain: '<S291>/Gain3' */
  rtb_Sum_gb = 0.1 * rtb_Divide2_f;

  /* BusCreator: '<S16>/Bus Creator' incorporates:
   *  Outport: '<Root>/out'
   *  RelationalOperator: '<S291>/Relational Operator'
   *  Sum: '<S291>/Add3'
   */
  Gen2_ref_Y->out.TJ_GasO[2] = (rtb_SumofElements_l > rtb_Divide2_f + rtb_Sum_gb);

  /* UnitDelay: '<S275>/Unit Delay2' */
  rtb_Gain6_jx = Gen2_ref_DWork->UnitDelay2_DSTATE_k;

  /* UnitDelay: '<S291>/Unit Delay2' */
  rtb_Sum_ig = Gen2_ref_DWork->UnitDelay2_DSTATE_p;

  /* Gain: '<S16>/W2kW1 ' */
  rtb_Divide2_f = 0.001 * Gen2_ref_B->Pd_filt_p.Switch;

  /* DataTypeConversion: '<S16>/Data Type Conversion16' */
  Gen2_ref_Y->out.Ptraj_SpeedCtrl = (real32_T)rtb_Divide2_f;

  /* BusCreator: '<Root>/Bus Creator' incorporates:
   *  BusCreator: '<S12>/Bus Creator'
   *  DataTypeConversion: '<S12>/Data Type Conversion'
   *  Outport: '<Root>/dbg'
   */
  Gen2_ref_Y->dbg.KeEstNetP.Ke_calc = (real32_T)r;

  /* Sum: '<S749>/Sum1' */
  r = rtb_Product1_c1_tmp;

  /* Gain: '<S749>/Gain7' */
  rtb_Divide2_f = -Gen2_ref_B->BusInput3.SpeedCtrl.rOutOfNWindow;

  /* Logic: '<S749>/Logical Operator4' incorporates:
   *  Logic: '<S749>/Logical Operator'
   *  Logic: '<S749>/Logical Operator1'
   *  Logic: '<S749>/Logical Operator2'
   *  Logic: '<S749>/Logical Operator3'
   *  MATLAB Function: '<S749>/MATLAB Function'
   *  RelationalOperator: '<S749>/Relational Operator'
   *  RelationalOperator: '<S749>/Relational Operator1'
   */
  rtb_LogicalOperator4_go = (rtb_Act && ((Gen2_ref_DWork->SR_LoadStep && (r >
    Gen2_ref_B->BusInput3.SpeedCtrl.rOutOfNWindow)) ||
    ((!Gen2_ref_DWork->SR_LoadStep) && (r < rtb_Divide2_f))));

  /* S-Function (sfix_look1_dyn): '<S431>/gain scheduling Keng' */
  /* Dynamic Look-Up Table Block: '<S431>/gain scheduling Keng'
   * Input0  Data Type:  Floating Point real_T
   * Input1  Data Type:  Floating Point real_T
   * Input2  Data Type:  Floating Point real_T
   * Output0 Data Type:  Floating Point real_T
   * Lookup Method: Linear_Endpoint
   *
   */
  LookUp_real_T_real_T( &(r), &rtb_Switch3_je[0], rtb_Gain3,
                       &Gen2_ref_B->BusInput3.SpeedCtrl.refPoint_iLQR_Keng_x[0],
                       12U, inst);

  /* Product: '<S431>/Product2' */
  rtb_Switch1_ep = r * rtb_Switch_nb;

  /* Switch: '<S13>/Switch' incorporates:
   *  DataTypeConversion: '<S12>/Data Type Conversion1'
   *  DataTypeConversion: '<S13>/Data Type Conversion'
   *  DataTypeConversion: '<S13>/Data Type Conversion1'
   *  DataTypeConversion: '<S431>/Data Type Conversion22'
   *  Gain: '<S13>/tom^3'
   *  Gain: '<S13>/tom^3_2'
   */
  if (rtb_LogicalOperator) {
    r = 1.0E-5 * (real32_T)Gen2_ref_B->Filter1_n.Switch;
  } else {
    r = 1.0E-5 * (real32_T)Gen2_ref_B->Filter1_o.Switch;
  }

  /* End of Switch: '<S13>/Switch' */

  /* Product: '<S13>/Product2' incorporates:
   *  Constant: '<S13>/4pi'
   */
  rtb_Switch_n = r * rtb_kW2W * Gen2_ref_B->T2s_filt.Switch * 12.566370614359172;

  /* Product: '<S13>/Product1' */
  r = rtb_dm_e_tmp * rtb_etaBreakConst;

  /* Abs: '<S856>/Abs' */
  rtb_Divide2_f = fabs(r);

  /* BusCreator: '<S16>/Bus Creator' incorporates:
   *  Constant: '<S5>/Constant2'
   *  Constant: '<S5>/Constant3'
   *  DataTypeConversion: '<S16>/Data Type Conversion'
   *  DataTypeConversion: '<S16>/Data Type Conversion11'
   *  DataTypeConversion: '<S16>/Data Type Conversion12'
   *  DataTypeConversion: '<S16>/Data Type Conversion13'
   *  DataTypeConversion: '<S16>/Data Type Conversion14'
   *  DataTypeConversion: '<S16>/Data Type Conversion15'
   *  DataTypeConversion: '<S16>/Data Type Conversion17'
   *  DataTypeConversion: '<S16>/Data Type Conversion18'
   *  DataTypeConversion: '<S16>/Data Type Conversion2'
   *  DataTypeConversion: '<S16>/Data Type Conversion3'
   *  DataTypeConversion: '<S16>/Data Type Conversion5'
   *  DataTypeConversion: '<S16>/Data Type Conversion6'
   *  DataTypeConversion: '<S16>/Data Type Conversion7'
   *  DataTypeConversion: '<S16>/Data Type Conversion8'
   *  Gain: '<S16>/Pa2bar'
   *  Logic: '<S275>/Logical Operator'
   *  Logic: '<S291>/Logical Operator'
   *  MATLAB Function: '<S715>/MATLAB Function1'
   *  Outport: '<Root>/out'
   *  RelationalOperator: '<S275>/Relational Operator1'
   *  RelationalOperator: '<S275>/Relational Operator2'
   *  RelationalOperator: '<S291>/Relational Operator1'
   *  RelationalOperator: '<S291>/Relational Operator2'
   *  SignalConversion generated from: '<S16>/Bus Creator'
   *  Sum: '<S275>/Add4'
   *  Sum: '<S275>/Add5'
   *  Sum: '<S291>/Add4'
   *  Sum: '<S291>/Add5'
   *  UnitDelay: '<S275>/Unit Delay'
   *  UnitDelay: '<S275>/Unit Delay1'
   *  UnitDelay: '<S275>/Unit Delay2'
   *  UnitDelay: '<S275>/Unit Delay3'
   *  UnitDelay: '<S291>/Unit Delay'
   *  UnitDelay: '<S291>/Unit Delay1'
   *  UnitDelay: '<S291>/Unit Delay2'
   *  UnitDelay: '<S291>/Unit Delay3'
   * */
  Gen2_ref_Y->out.rmdot_gas = (real32_T)rtb_Switch_g[0];
  Gen2_ref_Y->out.rmdot_gas_M = (real32_T)rtb_Switch_g[1];
  Gen2_ref_Y->out.rLamGen2 = (real32_T)rtb_Switch_g[2];
  Gen2_ref_Y->out.rPos_TV = (real32_T)rtb_Switch_g[3];
  Gen2_ref_Y->out.rPos_CBV = (real32_T)rtb_Switch_g[4];
  Gen2_ref_Y->out.rPos_WGV = (real32_T)rtb_Switch_g[5];
  Gen2_ref_Y->out.rPr_p2s_des = (real32_T)(1.0E-5 * rtb_Pa2bar_o);
  Gen2_ref_Y->out.rPrP2sLEANOXref = (real32_T)rtb_Sum_e;
  Gen2_ref_Y->out.rLamLimUp = (real32_T)rtb_Switch2_n5;
  Gen2_ref_Y->out.rLamLimLo = (real32_T)rtb_Switch1_k;
  Gen2_ref_Y->out.rLamss = (real32_T)rtb_PactOut_o;
  for (i = 0; i < 13; i++) {
    /* Switch: '<Root>/GasStop8' incorporates:
     *  DataTypeConversion: '<S16>/Data Type Conversion19'
     */
    if (rtb_bTV_sat) {
      Gen2_ref_Y->out.rKengMap[i] = (real32_T)
        Gen2_ref_B->sf_MATLABFunction1_l.y_map_new[i];
    } else {
      Gen2_ref_Y->out.rKengMap[i] = (real32_T)rtb_Switch3_je[i];
    }
```
